// eDataMappingVarNames.Router_Mobile_ModemState: 				st_Variable:= IotExtractType(monitor.Router.Mobile.ModemState, 0, 0); 
// eDataMappingVarNames.Router_Mobile_NetworkState: 				st_Variable:= IotExtractType(monitor.Router.Mobile.NetworkState, 0, 0); 
// eDataMappingVarNames.Router_Mobile_ui_ActiveSim: 				st_Variable:= IotExtractType(monitor.Router.Mobile.ui_ActiveSim, 0, 0); 
// eDataMappingVarNames.Router_Mobile_SimStatus: 				st_Variable:= IotExtractType(monitor.Router.Mobile.SimStatus, 0, 0); 
// eDataMappingVarNames.Router_Wifi_WifiClienModeStatus: 				st_Variable:= IotExtractType(monitor.Router.Wifi.WifiClienModeStatus, 0, 0); 
// eDataMappingVarNames.Router_Wifi_WifiAPModeStatus: 				st_Variable:= IotExtractType(monitor.Router.Wifi.WifiAPModeStatus, 0, 0); 
// eDataMappingVarNames.Router_Wifi_WifiApNumberOfClients: 				st_Variable:= IotExtractType(monitor.Router.Wifi.WifiApNumberOfClients, 0, 0); 
// eDataMappingVarNames.Router_e_SMSStatus: 				st_Variable:= IotExtractType(monitor.Router.e_SMSStatus, 0, 0); 
// eDataMappingVarNames.Router_Events_b_MBCommWarning: 				st_Variable:= IotExtractType(monitor.Router.Events.b_MBCommWarning, 0, 0); 
// eDataMappingVarNames.Router_Events_b_NoSimWarning: 				st_Variable:= IotExtractType(monitor.Router.Events.b_NoSimWarning, 0, 0); 
// eDataMappingVarNames.Router_Events_b_NoNetworkWarning: 				st_Variable:= IotExtractType(monitor.Router.Events.b_NoNetworkWarning, 0, 0); 
// eDataMappingVarNames.Router_Events_b_noGPSFixWarning: 				st_Variable:= IotExtractType(monitor.Router.Events.b_noGPSFixWarning, 0, 0); 
// eDataMappingVarNames.Router_Events_b_SMSNotSendError: 				st_Variable:= IotExtractType(monitor.Router.Events.b_SMSNotSendError, 0, 0); 
// eDataMappingVarNames.Router_Events_b_NoSMSNumberAvailable: 				st_Variable:= IotExtractType(monitor.Router.Events.b_NoSMSNumberAvailable, 0, 0); 
// eDataMappingVarNames.Router_Events_b_TimeUpdateFailed: 				st_Variable:= IotExtractType(monitor.Router.Events.b_TimeUpdateFailed, 0, 0); 
// eDataMappingVarNames.controlfb_control_b_start: 															st_Variable:= IotExtractType(controlvars.control.b_start, 0, 0); 
// eDataMappingVarNames.controlfb_control_b_stop: 																st_Variable:= IotExtractType(controlvars.control.b_stop, 0, 0); 
// eDataMappingVarNames.controlfb_control_b_shutdown: 															st_Variable:= IotExtractType(controlvars.control.b_shutdown, 0, 0); 
// eDataMappingVarNames.controlfb_control_b_Reset: 															st_Variable:= IotExtractType(controlvars.control.b_Reset, 0, 0); 
// eDataMappingVarNames.controlfb_control_b_SystemShutdown: 													st_Variable:= IotExtractType(controlvars.control.b_SystemShutdown, 0, 0); 
// eDataMappingVarNames.controlfb_control_b_EMstop: 															st_Variable:= IotExtractType(controlvars.control.b_EMstop, 0, 0); 
// eDataMappingVarNames.controlfb_control_b_ClearHistory: 														st_Variable:= IotExtractType(controlvars.control.b_ClearHistory, 0, 0); 
// eDataMappingVarNames.controlfb_control_b_ActivateSettings: 													st_Variable:= IotExtractType(controlvars.control.b_ActivateSettings, 0, 0); 
// eDataMappingVarNames.controlfb_control_b_startDeHum: 														st_Variable:= IotExtractType(controlvars.control.b_startDeHum, 0, 0); 
// eDataMappingVarNames.controlfb_Operation_inputgrid_b_SyncClose: 											st_Variable:= IotExtractType(controlvars.Operation.inputgrid.b_SyncClose, 0, 0); 
// eDataMappingVarNames.controlfb_Operation_Genset_b_manualStart: 												st_Variable:= IotExtractType(controlvars.Operation.Genset.b_manualStart, 0, 0); 
// eDataMappingVarNames.controlfb_Operation_PSB_b_SyncClose: 													st_Variable:= IotExtractType(controlvars.Operation.PSB.b_SyncClose, 0, 0); 
// eDataMappingVarNames.controlfb_Operation_charger_b_StartCharging: 											st_Variable:= IotExtractType(controlvars.Operation.charger.b_StartCharging, 0, 0); 
// eDataMappingVarNames.controlfb_Operation_charger_b_ResetCharger: 											st_Variable:= IotExtractType(controlvars.Operation.charger.b_ResetCharger, 0, 0); 
// eDataMappingVarNames.controlfb_Operation_system_r_NominalVoltage: 											st_Variable:= IotExtractType(controlvars.Operation.system.r_NominalVoltage, 0, 0); 
// eDataMappingVarNames.controlfb_Operation_system_r_NominalFrequency: 										st_Variable:= IotExtractType(controlvars.Operation.system.r_NominalFrequency, 0, 0); 
// eDataMappingVarNames.controlfb_Operation_system_r_Pset: 													st_Variable:= IotExtractType(controlvars.Operation.system.r_Pset, 0, 0); 
// eDataMappingVarNames.controlfb_Operation_system_r_Qset: 													st_Variable:= IotExtractType(controlvars.Operation.system.r_Qset, 0, 0); 
// eDataMappingVarNames.controlfb_Operation_system_r_PFset: 													st_Variable:= IotExtractType(controlvars.Operation.system.r_PFset, 0, 0); 
// eDataMappingVarNames.controlfb_Operation_system_b_PFsetEnable: 												st_Variable:= IotExtractType(controlvars.Operation.system.b_PFsetEnable, 0, 0); 
// eDataMappingVarNames.controlfb_Operation_system_b_SounderMute: 												st_Variable:= IotExtractType(controlvars.Operation.system.b_SounderMute, 0, 0); 
// eDataMappingVarNames.controlfb_Operation_system_b_SounderTest: 												st_Variable:= IotExtractType(controlvars.Operation.system.b_SounderTest, 0, 0); 
// eDataMappingVarNames.controlfb_Operation_system_b_GenGridModeTrans: 										st_Variable:= IotExtractType(controlvars.Operation.system.b_GenGridModeTrans, 0, 0); 
// eDataMappingVarNames.controlfb_Operation_system_b_GridTakeOverEnable: 										st_Variable:= IotExtractType(controlvars.Operation.system.b_GridTakeOverEnable, 0, 0); 
// eDataMappingVarNames.controlfb_Operation_parallel_b_DetectSlaves: 											st_Variable:= IotExtractType(controlvars.Operation.parallel.b_DetectSlaves, 0, 0); 
// eDataMappingVarNames.controlfb_Operation_parallel_r_ActivePowerSlave1: 										st_Variable:= IotExtractType(controlvars.Operation.parallel.r_ActivePowerSlave1, 0, 0); 
// eDataMappingVarNames.controlfb_Operation_parallel_r_ReactivePowerSlave1: 									st_Variable:= IotExtractType(controlvars.Operation.parallel.r_ReactivePowerSlave1, 0, 0); 
// eDataMappingVarNames.controlfb_Operation_parallel_r_ActivePowerSlave2: 										st_Variable:= IotExtractType(controlvars.Operation.parallel.r_ActivePowerSlave2, 0, 0); 
// eDataMappingVarNames.controlfb_Operation_parallel_r_ReactivePowerSlave2: 									st_Variable:= IotExtractType(controlvars.Operation.parallel.r_ReactivePowerSlave2, 0, 0); 
// eDataMappingVarNames.controlfb_Operation_BMS_b_ManualStartHVDC: 											st_Variable:= IotExtractType(controlvars.Operation.BMS.b_ManualStartHVDC, 0, 0); 
// eDataMappingVarNames.controlfb_SoftSettings_inputgrid_PeakshaveMode: 										st_Variable:= IotExtractType(controlvars.SoftSettings.inputgrid.PeakshaveMode, 0, 0); 
// eDataMappingVarNames.controlfb_SoftSettings_inputgrid_setpointTimeslot1_r_SocTarget:		 				st_Variable:= IotExtractType(controlvars.SoftSettings.inputgrid.setpointTimeslot1.r_SocTarget, 0, 0); 
// eDataMappingVarNames.controlfb_SoftSettings_inputgrid_setpointTimeslot1_r_IdleChargePower: 					st_Variable:= IotExtractType(controlvars.SoftSettings.inputgrid.setpointTimeslot1.r_IdleChargePower, 0, 0); 
// eDataMappingVarNames.controlfb_SoftSettings_inputgrid_setpointTimeslot1_r_FeedInCurrentLimitSoft: 			st_Variable:= IotExtractType(controlvars.SoftSettings.inputgrid.setpointTimeslot1.r_FeedInCurrentLimitSoft, 0, 0); 
// eDataMappingVarNames.controlfb_SoftSettings_inputgrid_setpointTimeslot1_r_SupplyCurrentLimitSoft: 			st_Variable:= IotExtractType(controlvars.SoftSettings.inputgrid.setpointTimeslot1.r_SupplyCurrentLimitSoft, 0, 0); 
// eDataMappingVarNames.controlfb_SoftSettings_inputgrid_setpointTimeslot2_r_SocTarget: 						st_Variable:= IotExtractType(controlvars.SoftSettings.inputgrid.setpointTimeslot2.r_SocTarget, 0, 0); 
// eDataMappingVarNames.controlfb_SoftSettings_inputgrid_setpointTimeslot2_r_IdleChargePower: 					st_Variable:= IotExtractType(controlvars.SoftSettings.inputgrid.setpointTimeslot2.r_IdleChargePower, 0, 0); 
// eDataMappingVarNames.controlfb_SoftSettings_inputgrid_setpointTimeslot2_r_FeedInCurrentLimitSoft: 			st_Variable:= IotExtractType(controlvars.SoftSettings.inputgrid.setpointTimeslot2.r_FeedInCurrentLimitSoft, 0, 0); 
// eDataMappingVarNames.controlfb_SoftSettings_inputgrid_setpointTimeslot2_r_SupplyCurrentLimitSoft: 			st_Variable:= IotExtractType(controlvars.SoftSettings.inputgrid.setpointTimeslot2.r_SupplyCurrentLimitSoft, 0, 0); 
// eDataMappingVarNames.controlfb_SoftSettings_inputgrid_b_BreakerControl: 									st_Variable:= IotExtractType(controlvars.SoftSettings.inputgrid.b_BreakerControl, 0, 0); 
// eDataMappingVarNames.controlfb_SoftSettings_inputgrid_b_ReverseCTDirection: 								st_Variable:= IotExtractType(controlvars.SoftSettings.inputgrid.b_ReverseCTDirection, 0, 0); 
// eDataMappingVarNames.controlfb_SoftSettings_inputgrid_ui_CTrange: 											st_Variable:= IotExtractType(controlvars.SoftSettings.inputgrid.ui_CTrange, 0, 0); 
// eDataMappingVarNames.controlfb_SoftSettings_inputgrid_r_VTratio: 											st_Variable:= IotExtractType(controlvars.SoftSettings.inputgrid.r_VTratio, 0, 0); 
// eDataMappingVarNames.controlfb_SoftSettings_inputgrid_b_GridCodesActive: 									st_Variable:= IotExtractType(controlvars.SoftSettings.inputgrid.b_GridCodesActive, 0, 0); 
// eDataMappingVarNames.controlfb_SoftSettings_inputgrid_b_WeakGridInput: 										st_Variable:= IotExtractType(controlvars.SoftSettings.inputgrid.b_WeakGridInput, 0, 0); 
// eDataMappingVarNames.controlfb_SoftSettings_inputgrid_breaker_AutoConnect: 									st_Variable:= IotExtractType(controlvars.SoftSettings.inputgrid.breaker.AutoConnect, 0, 0); 
// eDataMappingVarNames.controlfb_SoftSettings_inputgrid_breaker_ShutdownDisconnect: 							st_Variable:= IotExtractType(controlvars.SoftSettings.inputgrid.breaker.ShutdownDisconnect, 0, 0); 
// eDataMappingVarNames.controlfb_SoftSettings_inputgrid_breaker_EMstopDisconnect: 							st_Variable:= IotExtractType(controlvars.SoftSettings.inputgrid.breaker.EMstopDisconnect, 0, 0); 
// eDataMappingVarNames.controlfb_SoftSettings_inputgrid_breaker_CurrentLimitDisconnect: 						st_Variable:= IotExtractType(controlvars.SoftSettings.inputgrid.breaker.CurrentLimitDisconnect, 0, 0); 
// eDataMappingVarNames.controlfb_SoftSettings_inputgrid_breaker_CurrentLimitRetries: 							st_Variable:= IotExtractType(controlvars.SoftSettings.inputgrid.breaker.CurrentLimitRetries, 0, 0); 
// eDataMappingVarNames.controlfb_SoftSettings_inputgenset_b_AutoStartStop: 									st_Variable:= IotExtractType(controlvars.SoftSettings.inputgenset.b_AutoStartStop, 0, 0); 
// eDataMappingVarNames.controlfb_SoftSettings_inputgenset_b_HydridMode: 										st_Variable:= IotExtractType(controlvars.SoftSettings.inputgenset.b_HydridMode, 0, 0); 
// eDataMappingVarNames.controlfb_SoftSettings_inputgenset_b_EnableSchedule: 									st_Variable:= IotExtractType(controlvars.SoftSettings.inputgenset.b_EnableSchedule, 0, 0); 
// eDataMappingVarNames.controlfb_SoftSettings_inputgenset_setpointTimeslot1_r_SoCStart: 						st_Variable:= IotExtractType(controlvars.SoftSettings.inputgenset.setpointTimeslot1.r_SoCStart, 0, 0); 
// eDataMappingVarNames.controlfb_SoftSettings_inputgenset_setpointTimeslot1_r_SoCStop: 						st_Variable:= IotExtractType(controlvars.SoftSettings.inputgenset.setpointTimeslot1.r_SoCStop, 0, 0); 
// eDataMappingVarNames.controlfb_SoftSettings_inputgenset_setpointTimeslot1_r_BatteryloadStart: 				st_Variable:= IotExtractType(controlvars.SoftSettings.inputgenset.setpointTimeslot1.r_BatteryloadStart, 0, 0); 
// eDataMappingVarNames.controlfb_SoftSettings_inputgenset_setpointTimeslot1_r_BatteryloadStop: 				st_Variable:= IotExtractType(controlvars.SoftSettings.inputgenset.setpointTimeslot1.r_BatteryloadStop, 0, 0); 
// eDataMappingVarNames.controlfb_SoftSettings_inputgenset_setpointTimeslot1_b_StartAtBatteryError: 			st_Variable:= IotExtractType(controlvars.SoftSettings.inputgenset.setpointTimeslot1.b_StartAtBatteryError, 0, 0); 
// eDataMappingVarNames.controlfb_SoftSettings_inputgenset_setpointTimeslot2_r_SoCStart: 						st_Variable:= IotExtractType(controlvars.SoftSettings.inputgenset.setpointTimeslot2.r_SoCStart, 0, 0); 
// eDataMappingVarNames.controlfb_SoftSettings_inputgenset_setpointTimeslot2_r_SoCStop: 						st_Variable:= IotExtractType(controlvars.SoftSettings.inputgenset.setpointTimeslot2.r_SoCStop, 0, 0); 
// eDataMappingVarNames.controlfb_SoftSettings_inputgenset_setpointTimeslot2_r_BatteryloadStart: 				st_Variable:= IotExtractType(controlvars.SoftSettings.inputgenset.setpointTimeslot2.r_BatteryloadStart, 0, 0); 
// eDataMappingVarNames.controlfb_SoftSettings_inputgenset_setpointTimeslot2_r_BatteryloadStop: 				st_Variable:= IotExtractType(controlvars.SoftSettings.inputgenset.setpointTimeslot2.r_BatteryloadStop, 0, 0); 
// eDataMappingVarNames.controlfb_SoftSettings_inputgenset_setpointTimeslot2_b_StartAtBatteryError: 			st_Variable:= IotExtractType(controlvars.SoftSettings.inputgenset.setpointTimeslot2.b_StartAtBatteryError, 0, 0); 
// eDataMappingVarNames.controlfb_SoftSettings_inputgenset_b_PSBExtGensetMonitoring: 							st_Variable:= IotExtractType(controlvars.SoftSettings.inputgenset.b_PSBExtGensetMonitoring, 0, 0); 
// eDataMappingVarNames.controlfb_SoftSettings_inputgenset_b_FreqProtectionEnable: 							st_Variable:= IotExtractType(controlvars.SoftSettings.inputgenset.b_FreqProtectionEnable, 0, 0); 
// eDataMappingVarNames.controlfb_SoftSettings_inputgenset_Generator_e_GensetMode: 							st_Variable:= IotExtractType(controlvars.SoftSettings.inputgenset.Generator.e_GensetMode, 0, 0); 
// eDataMappingVarNames.controlfb_SoftSettings_inputgenset_Generator_b_GensetLoadshareLine: 					st_Variable:= IotExtractType(controlvars.SoftSettings.inputgenset.Generator.b_GensetLoadshareLine, 0, 0); 
// eDataMappingVarNames.controlfb_SoftSettings_inputgenset_Generator_r_RatedPower: 							st_Variable:= IotExtractType(controlvars.SoftSettings.inputgenset.Generator.r_RatedPower, 0, 0); 
// eDataMappingVarNames.controlfb_SoftSettings_inputgenset_Generator_r_powerloadMax: 							st_Variable:= IotExtractType(controlvars.SoftSettings.inputgenset.Generator.r_powerloadMax, 0, 0); 
// eDataMappingVarNames.controlfb_SoftSettings_inputgenset_Generator_r_PowerloadMin: 							st_Variable:= IotExtractType(controlvars.SoftSettings.inputgenset.Generator.r_PowerloadMin, 0, 0); 
// eDataMappingVarNames.controlfb_SoftSettings_inputgenset_Generator_r_PowerloadEff: 							st_Variable:= IotExtractType(controlvars.SoftSettings.inputgenset.Generator.r_PowerloadEff, 0, 0); 
// eDataMappingVarNames.controlfb_SoftSettings_inputgenset_Generator_r_ramprate: 								st_Variable:= IotExtractType(controlvars.SoftSettings.inputgenset.Generator.r_ramprate, 0, 0); 
// eDataMappingVarNames.controlfb_SoftSettings_inputgenset_Generator_ui_CooldownTime: 							st_Variable:= IotExtractType(controlvars.SoftSettings.inputgenset.Generator.ui_CooldownTime, 0, 0); 
// eDataMappingVarNames.controlfb_SoftSettings_inputgenset_Generator_ui_WarmupTime: 							st_Variable:= IotExtractType(controlvars.SoftSettings.inputgenset.Generator.ui_WarmupTime, 0, 0); 
// eDataMappingVarNames.controlfb_SoftSettings_inputgenset_Loadbank_b_Enable: 									st_Variable:= IotExtractType(controlvars.SoftSettings.inputgenset.Loadbank.b_Enable, 0, 0); 
// eDataMappingVarNames.controlfb_SoftSettings_inputgenset_Loadbank_r_PowerRating: 							st_Variable:= IotExtractType(controlvars.SoftSettings.inputgenset.Loadbank.r_PowerRating, 0, 0); 
// eDataMappingVarNames.controlfb_SoftSettings_inputgenset_Loadbank_r_PowerStepSize: 							st_Variable:= IotExtractType(controlvars.SoftSettings.inputgenset.Loadbank.r_PowerStepSize, 0, 0); 
// eDataMappingVarNames.controlfb_SoftSettings_PSB_PeakshaveMode: 												st_Variable:= IotExtractType(controlvars.SoftSettings.PSB.PeakshaveMode, 0, 0); 
// eDataMappingVarNames.controlfb_SoftSettings_PSB_setpointTimeslot1_r_SocTarget: 								st_Variable:= IotExtractType(controlvars.SoftSettings.PSB.setpointTimeslot1.r_SocTarget, 0, 0); 
// eDataMappingVarNames.controlfb_SoftSettings_PSB_setpointTimeslot1_r_IdleChargePower: 						st_Variable:= IotExtractType(controlvars.SoftSettings.PSB.setpointTimeslot1.r_IdleChargePower, 0, 0); 
// eDataMappingVarNames.controlfb_SoftSettings_PSB_setpointTimeslot1_r_FeedInCurrentLimitSoft: 				st_Variable:= IotExtractType(controlvars.SoftSettings.PSB.setpointTimeslot1.r_FeedInCurrentLimitSoft, 0, 0); 
// eDataMappingVarNames.controlfb_SoftSettings_PSB_setpointTimeslot1_r_SupplyCurrentLimitSoft: 				st_Variable:= IotExtractType(controlvars.SoftSettings.PSB.setpointTimeslot1.r_SupplyCurrentLimitSoft, 0, 0); 
// eDataMappingVarNames.controlfb_SoftSettings_PSB_setpointTimeslot2_r_SocTarget: 								st_Variable:= IotExtractType(controlvars.SoftSettings.PSB.setpointTimeslot2.r_SocTarget, 0, 0); 
// eDataMappingVarNames.controlfb_SoftSettings_PSB_setpointTimeslot2_r_IdleChargePower: 						st_Variable:= IotExtractType(controlvars.SoftSettings.PSB.setpointTimeslot2.r_IdleChargePower, 0, 0); 
// eDataMappingVarNames.controlfb_SoftSettings_PSB_setpointTimeslot2_r_FeedInCurrentLimitSoft: 				st_Variable:= IotExtractType(controlvars.SoftSettings.PSB.setpointTimeslot2.r_FeedInCurrentLimitSoft, 0, 0); 
// eDataMappingVarNames.controlfb_SoftSettings_PSB_setpointTimeslot2_r_SupplyCurrentLimitSoft: 				st_Variable:= IotExtractType(controlvars.SoftSettings.PSB.setpointTimeslot2.r_SupplyCurrentLimitSoft, 0, 0); 
// eDataMappingVarNames.controlfb_SoftSettings_PSB_b_BreakerControl: 											st_Variable:= IotExtractType(controlvars.SoftSettings.PSB.b_BreakerControl, 0, 0); 
// eDataMappingVarNames.controlfb_SoftSettings_PSB_b_ReverseCTDirection: 										st_Variable:= IotExtractType(controlvars.SoftSettings.PSB.b_ReverseCTDirection, 0, 0); 
// eDataMappingVarNames.controlfb_SoftSettings_PSB_ui_CTrange: 												st_Variable:= IotExtractType(controlvars.SoftSettings.PSB.ui_CTrange, 0, 0); 
// eDataMappingVarNames.controlfb_SoftSettings_PSB_r_VTratio: 													st_Variable:= IotExtractType(controlvars.SoftSettings.PSB.r_VTratio, 0, 0); 
// eDataMappingVarNames.controlfb_SoftSettings_system_b_EnableSchedule: 										st_Variable:= IotExtractType(controlvars.SoftSettings.system.b_EnableSchedule, 0, 0); 
// eDataMappingVarNames.controlfb_SoftSettings_system_b_EnableTransportMode: 									st_Variable:= IotExtractType(controlvars.SoftSettings.system.b_EnableTransportMode, 0, 0); 
// eDataMappingVarNames.controlfb_SoftSettings_system_b_EcoModeEnable: 										st_Variable:= IotExtractType(controlvars.SoftSettings.system.b_EcoModeEnable, 0, 0); 
// eDataMappingVarNames.controlfb_SoftSettings_system_e_UgridPowerMode: 										st_Variable:= IotExtractType(controlvars.SoftSettings.system.e_UgridPowerMode, 0, 0); 
// eDataMappingVarNames.controlfb_SoftSettings_system_e_NetcontactorMode: 										st_Variable:= IotExtractType(controlvars.SoftSettings.system.e_NetcontactorMode, 0, 0); 
// eDataMappingVarNames.controlfb_SoftSettings_system_e_UgridPowerLimitingMode: 								st_Variable:= IotExtractType(controlvars.SoftSettings.system.e_UgridPowerLimitingMode, 0, 0); 
// eDataMappingVarNames.controlfb_SoftSettings_system_b_AutomaticSwitching: 									st_Variable:= IotExtractType(controlvars.SoftSettings.system.b_AutomaticSwitching, 0, 0); 
// eDataMappingVarNames.controlfb_SoftSettings_system_b_AMF: 													st_Variable:= IotExtractType(controlvars.SoftSettings.system.b_AMF, 0, 0); 
// eDataMappingVarNames.controlfb_SoftSettings_system_r_FrequencyDroop: 										st_Variable:= IotExtractType(controlvars.SoftSettings.system.r_FrequencyDroop, 0, 0); 
// eDataMappingVarNames.controlfb_SoftSettings_system_r_VoltageDroop: 											st_Variable:= IotExtractType(controlvars.SoftSettings.system.r_VoltageDroop, 0, 0); 
// eDataMappingVarNames.controlfb_SoftSettings_system_r_SocMin: 												st_Variable:= IotExtractType(controlvars.SoftSettings.system.r_SocMin, 0, 0); 
// eDataMappingVarNames.controlfb_SoftSettings_system_r_SocMax: 												st_Variable:= IotExtractType(controlvars.SoftSettings.system.r_SocMax, 0, 0); 
// eDataMappingVarNames.controlfb_SoftSettings_system_r_PDischargeLimit: 										st_Variable:= IotExtractType(controlvars.SoftSettings.system.r_PDischargeLimit, 0, 0); 
// eDataMappingVarNames.controlfb_SoftSettings_system_r_PChargeLimit: 											st_Variable:= IotExtractType(controlvars.SoftSettings.system.r_PChargeLimit, 0, 0); 
// eDataMappingVarNames.controlfb_SoftSettings_system_r_AMax: 													st_Variable:= IotExtractType(controlvars.SoftSettings.system.r_AMax, 0, 0); 
// eDataMappingVarNames.controlfb_SoftSettings_system_s_SystemName: 											st_Variable:= IotExtractType(controlvars.SoftSettings.system.s_SystemName, 0, 0); 
// eDataMappingVarNames.controlfb_SoftSettings_system_s_SMSnumber: 											st_Variable:= IotExtractType(controlvars.SoftSettings.system.s_SMSnumber, 0, 0); 
// eDataMappingVarNames.controlfb_SoftSettings_system_ScheduleTimeSlot1_b_active: 								st_Variable:= IotExtractType(controlvars.SoftSettings.system.ScheduleTimeSlot1.b_active, 0, 0); 
// eDataMappingVarNames.controlfb_SoftSettings_system_ScheduleTimeSlot1_usi_DayOfWeek: 						st_Variable:= IotExtractType(controlvars.SoftSettings.system.ScheduleTimeSlot1.usi_DayOfWeek, 0, 0); 
// eDataMappingVarNames.controlfb_SoftSettings_system_ScheduleTimeSlot1_usi_HourOfDay: 						st_Variable:= IotExtractType(controlvars.SoftSettings.system.ScheduleTimeSlot1.usi_HourOfDay, 0, 0); 
// eDataMappingVarNames.controlfb_SoftSettings_system_ScheduleTimeSlot1_usi_MinuteOfHour: 						st_Variable:= IotExtractType(controlvars.SoftSettings.system.ScheduleTimeSlot1.usi_MinuteOfHour, 0, 0); 
// eDataMappingVarNames.controlfb_SoftSettings_system_ScheduleTimeSlot2_b_active: 								st_Variable:= IotExtractType(controlvars.SoftSettings.system.ScheduleTimeSlot2.b_active, 0, 0); 
// eDataMappingVarNames.controlfb_SoftSettings_system_ScheduleTimeSlot2_usi_DayOfWeek: 						st_Variable:= IotExtractType(controlvars.SoftSettings.system.ScheduleTimeSlot2.usi_DayOfWeek, 0, 0); 
// eDataMappingVarNames.controlfb_SoftSettings_system_ScheduleTimeSlot2_usi_HourOfDay: 						st_Variable:= IotExtractType(controlvars.SoftSettings.system.ScheduleTimeSlot2.usi_HourOfDay, 0, 0); 
// eDataMappingVarNames.controlfb_SoftSettings_system_ScheduleTimeSlot2_usi_MinuteOfHour: 						st_Variable:= IotExtractType(controlvars.SoftSettings.system.ScheduleTimeSlot2.usi_MinuteOfHour, 0, 0); 
// eDataMappingVarNames.controlfb_SoftSettings_system_by_LEDbrightness: 										st_Variable:= IotExtractType(controlvars.SoftSettings.system.by_LEDbrightness, 0, 0); 
// eDataMappingVarNames.controlfb_SoftSettings_setup_e_AcInputType: 											st_Variable:= IotExtractType(controlvars.SoftSettings.setup.e_AcInputType, 0, 0); 
// eDataMappingVarNames.controlfb_SoftSettings_setup_b_MasterSlaveMode: 										st_Variable:= IotExtractType(controlvars.SoftSettings.setup.b_MasterSlaveMode, 0, 0); 
// eDataMappingVarNames.controlfb_SoftSettings_setup_b_PeakshaveBoxEnable: 									st_Variable:= IotExtractType(controlvars.SoftSettings.setup.b_PeakshaveBoxEnable, 0, 0); 
// eDataMappingVarNames.controlfb_SoftSettings_setup_e_Gridmode: 												st_Variable:= IotExtractType(controlvars.SoftSettings.setup.e_Gridmode, 0, 0); 
// eDataMappingVarNames.controlfb_SoftSettings_setup_e_DcCouplingType: 										st_Variable:= IotExtractType(controlvars.SoftSettings.setup.e_DcCouplingType, 0, 0); 
// eDataMappingVarNames.controlfb_SoftSettings_setup_b_ExtGenset: 												st_Variable:= IotExtractType(controlvars.SoftSettings.setup.b_ExtGenset, 0, 0); 
// eDataMappingVarNames.controlfb_HardSettings_setup_e_ControlSource: 											st_Variable:= IotExtractType(controlvars.HardSettings.setup.e_ControlSource, 0, 0); 
// eDataMappingVarNames.controlfb_HardSettings_charger_r_PowerMax: 											st_Variable:= IotExtractType(controlvars.HardSettings.charger.r_PowerMax, 0, 0); 
// eDataMappingVarNames.controlfb_HardSettings_parallel_b_MasterSlaveEnabled: 									st_Variable:= IotExtractType(controlvars.HardSettings.parallel.b_MasterSlaveEnabled, 0, 0); 
// eDataMappingVarNames.controlfb_HardSettings_parallel_b_UnitIsMaster: 										st_Variable:= IotExtractType(controlvars.HardSettings.parallel.b_UnitIsMaster, 0, 0); 
// eDataMappingVarNames.controlfb_HardSettings_parallel_b_ShutdownOnCommError: 								st_Variable:= IotExtractType(controlvars.HardSettings.parallel.b_ShutdownOnCommError, 0, 0); 
// eDataMappingVarNames.controlfb_HardSettings_parallel_b_EffiencyMode: 										st_Variable:= IotExtractType(controlvars.HardSettings.parallel.b_EffiencyMode, 0, 0); 
// eDataMappingVarNames.controlfb_HardSettings_parallel_r_VoltageDroop: 										st_Variable:= IotExtractType(controlvars.HardSettings.parallel.r_VoltageDroop, 0, 0); 
// eDataMappingVarNames.controlfb_HardSettings_parallel_r_FrequencyDroop: 										st_Variable:= IotExtractType(controlvars.HardSettings.parallel.r_FrequencyDroop, 0, 0); 
// eDataMappingVarNames.controlfb_HardSettings_system_r_PDischargeLimit: 										st_Variable:= IotExtractType(controlvars.HardSettings.system.r_PDischargeLimit, 0, 0); 
// eDataMappingVarNames.controlfb_HardSettings_system_r_PChargeLimit: 											st_Variable:= IotExtractType(controlvars.HardSettings.system.r_PChargeLimit, 0, 0); 
// eDataMappingVarNames.controlfb_HardSettings_system_r_SMax: 													st_Variable:= IotExtractType(controlvars.HardSettings.system.r_SMax, 0, 0); 
// eDataMappingVarNames.controlfb_HardSettings_system_r_Amax: 													st_Variable:= IotExtractType(controlvars.HardSettings.system.r_Amax, 0, 0); 
// eDataMappingVarNames.controlfb_HardSettings_system_e_EarthingSystem: 										st_Variable:= IotExtractType(controlvars.HardSettings.system.e_EarthingSystem, 0, 0); 
// eDataMappingVarNames.controlfb_HardSettings_system_a_ui_InputCurrentLimit_1: 								st_Variable:= IotExtractType(controlvars.HardSettings.system.a_ui_InputCurrentLimit[1], 0, 0); 
// eDataMappingVarNames.controlfb_HardSettings_system_a_ui_InputCurrentLimit_2: 								st_Variable:= IotExtractType(controlvars.HardSettings.system.a_ui_InputCurrentLimit[2], 0, 0); 
// eDataMappingVarNames.controlfb_HardSettings_system_a_ui_OutputCurrentLimit_1: 								st_Variable:= IotExtractType(controlvars.HardSettings.system.a_ui_OutputCurrentLimit[1], 0, 0); 
// eDataMappingVarNames.controlfb_HardSettings_system_a_ui_OutputCurrentLimit_2: 								st_Variable:= IotExtractType(controlvars.HardSettings.system.a_ui_OutputCurrentLimit[2], 0, 0); 
// eDataMappingVarNames.controlfb_HardSettings_system_a_ui_OutputCurrentLimit_3: 								st_Variable:= IotExtractType(controlvars.HardSettings.system.a_ui_OutputCurrentLimit[3], 0, 0); 
// eDataMappingVarNames.Generator_CommunicationOK: 				st_Variable:= IotExtractType(monitor.Generator.CommunicationOK, 0, 0); 
// eDataMappingVarNames.Generator_FuelLow: 				st_Variable:= IotExtractType(monitor.Generator.FuelLow, 0, 0); 
// eDataMappingVarNames.Generator_FuelCritical: 				st_Variable:= IotExtractType(monitor.Generator.FuelCritical, 0, 0); 
// eDataMappingVarNames.Generator_bGenBreakerClosed: 				st_Variable:= IotExtractType(monitor.Generator.bGenBreakerClosed, 0, 0); 
// eDataMappingVarNames.Generator_bMainBreakerClosed: 				st_Variable:= IotExtractType(monitor.Generator.bMainBreakerClosed, 0, 0); 
// eDataMappingVarNames.Generator_bGenRunning: 				st_Variable:= IotExtractType(monitor.Generator.bGenRunning, 0, 0); 
// eDataMappingVarNames.Generator_bGenVoltFreqOK: 				st_Variable:= IotExtractType(monitor.Generator.bGenVoltFreqOK, 0, 0); 
// eDataMappingVarNames.Generator_bMainsFailure: 				st_Variable:= IotExtractType(monitor.Generator.bMainsFailure, 0, 0); 
// eDataMappingVarNames.Generator_eActiveGenMode: 				st_Variable:= IotExtractType(monitor.Generator.eActiveGenMode, 0, 0); 
// eDataMappingVarNames.Generator_bIslandModeActive: 				st_Variable:= IotExtractType(monitor.Generator.bIslandModeActive, 0, 0); 
// eDataMappingVarNames.Generator_bAMFActive: 				st_Variable:= IotExtractType(monitor.Generator.bAMFActive, 0, 0); 
// eDataMappingVarNames.Generator_bPeakshaveActive: 				st_Variable:= IotExtractType(monitor.Generator.bPeakshaveActive, 0, 0); 
// eDataMappingVarNames.Generator_bFixedPowerActive: 				st_Variable:= IotExtractType(monitor.Generator.bFixedPowerActive, 0, 0); 
// eDataMappingVarNames.Generator_ar_LineVoltage_AVG: 				st_Variable:= IotExtractType(monitor.Generator.ar_LineVoltage[0], 1, 1); 
// eDataMappingVarNames.Generator_ar_LineVoltage_L1: 				st_Variable:= IotExtractType(monitor.Generator.ar_LineVoltage[1], 1, 1); 
// eDataMappingVarNames.Generator_ar_LineVoltage_L2: 				st_Variable:= IotExtractType(monitor.Generator.ar_LineVoltage[2], 1, 1); 
// eDataMappingVarNames.Generator_ar_LineVoltage_L3: 				st_Variable:= IotExtractType(monitor.Generator.ar_LineVoltage[3], 1, 1); 
// eDataMappingVarNames.Generator_ar_PhaseVoltage_AVG: 				st_Variable:= IotExtractType(monitor.Generator.ar_PhaseVoltage[0], 1, 1); 
// eDataMappingVarNames.Generator_ar_PhaseVoltage_L1: 				st_Variable:= IotExtractType(monitor.Generator.ar_PhaseVoltage[1], 1, 1); 
// eDataMappingVarNames.Generator_ar_PhaseVoltage_L2: 				st_Variable:= IotExtractType(monitor.Generator.ar_PhaseVoltage[2], 1, 1); 
// eDataMappingVarNames.Generator_ar_PhaseVoltage_L3: 				st_Variable:= IotExtractType(monitor.Generator.ar_PhaseVoltage[3], 1, 1); 
// eDataMappingVarNames.Generator_ar_Frequency_AVG: 				st_Variable:= IotExtractType(monitor.Generator.ar_Frequency[0], 2, 1); 
// eDataMappingVarNames.Generator_ar_Frequency_L1: 				st_Variable:= IotExtractType(monitor.Generator.ar_Frequency[1], 2, 1); 
// eDataMappingVarNames.Generator_ar_Frequency_L2: 				st_Variable:= IotExtractType(monitor.Generator.ar_Frequency[2], 2, 1); 
// eDataMappingVarNames.Generator_ar_Frequency_L3: 				st_Variable:= IotExtractType(monitor.Generator.ar_Frequency[3], 2, 1); 
// eDataMappingVarNames.Generator_ar_Current_AVG: 				st_Variable:= IotExtractType(monitor.Generator.ar_Current[0], 1, 1); 
// eDataMappingVarNames.Generator_ar_Current_L1: 				st_Variable:= IotExtractType(monitor.Generator.ar_Current[1], 1, 1); 
// eDataMappingVarNames.Generator_ar_Current_L2: 				st_Variable:= IotExtractType(monitor.Generator.ar_Current[2], 1, 1); 
// eDataMappingVarNames.Generator_ar_Current_L3: 				st_Variable:= IotExtractType(monitor.Generator.ar_Current[3], 1, 1); 
// eDataMappingVarNames.Generator_ar_PowerFactor_AVG: 				st_Variable:= IotExtractType(monitor.Generator.ar_PowerFactor[0], 2, 0); 
// eDataMappingVarNames.Generator_ar_ActivePower_AVG: 				st_Variable:= IotExtractType(monitor.Generator.ar_ActivePower[0], 1, 1); 
// eDataMappingVarNames.Generator_ar_ActivePower_L1: 				st_Variable:= IotExtractType(monitor.Generator.ar_ActivePower[1], 1, 1); 
// eDataMappingVarNames.Generator_ar_ActivePower_L2: 				st_Variable:= IotExtractType(monitor.Generator.ar_ActivePower[2], 1, 1); 
// eDataMappingVarNames.Generator_ar_ActivePower_L3: 				st_Variable:= IotExtractType(monitor.Generator.ar_ActivePower[3], 1, 1); 
// eDataMappingVarNames.Generator_ar_ReactivePower_AVG: 				st_Variable:= IotExtractType(monitor.Generator.ar_ReactivePower[0], 1, 1); 
// eDataMappingVarNames.Generator_ar_ApparentPower_AVG: 				st_Variable:= IotExtractType(monitor.Generator.ar_ApparentPower[0], 1, 1); 
// eDataMappingVarNames.HartingIO_b_DigitalInput1Active: 				st_Variable:= IotExtractType(monitor.HartingIO.b_DigitalInput1Active, 0, 0); 
// eDataMappingVarNames.HartingIO_b_DigitalInput2Active: 				st_Variable:= IotExtractType(monitor.HartingIO.b_DigitalInput2Active, 0, 0); 
// eDataMappingVarNames.HartingIO_b_GenLowFuel: 				st_Variable:= IotExtractType(monitor.HartingIO.b_GenLowFuel, 0, 0); 
// eDataMappingVarNames.HartingIO_b_ExtSystemShutdownRequest: 				st_Variable:= IotExtractType(monitor.HartingIO.b_ExtSystemShutdownRequest, 0, 0); 
// eDataMappingVarNames.HartingIO_b_ExtEMstopOK: 				st_Variable:= IotExtractType(monitor.HartingIO.b_ExtEMstopOK, 0, 0); 
// eDataMappingVarNames.HartingIO_b_ExtEMstopActive: 				st_Variable:= IotExtractType(monitor.HartingIO.b_ExtEMstopActive, 0, 0); 
END_CASE

IF index >= eDataMappingVarNames.controlfb_control_b_start AND index <= eDataMappingVarNames.controlfb_HardSettings_system_a_ui_OutputCurrentLimit_3 THEN
	st_RW.ReadFromNUC := aData[index].LogType <> 0;
	st_RW.WriteToNUC := FALSE;
ELSE
	st_RW.ReadFromNUC := FALSE;
	st_RW.WriteToNUC :=  aData[index].LogType <> 0;
END_IF


//-------------------------------Write to output---------------------------------------------
IotMappingV2.sName		:= aData[index].Label;				//Name of the variable
IotMappingV2.sValue		:= st_Variable.sValue;	//Extracted value of the variable
IotMappingV2.eUpdate	:= aData[index].LogInterval;				//Update frequency
IotMappingV2.st_RW		:= st_RW;				//Read/Write
IotMappingV2.pAdress	:= st_Variable.pAdress; //Adress pointer to variable
IotMappingV2.diSize		:= st_Variable.diSize;
IotMappingV2.ClassType	:= st_Variable.ClassType; //Extracted data type of the variable
IotMappingV2.bNumber	:= st_Variable.bNumber;
IotMappingV2.bJson		:= bJson;
END_METHOD

METHOD IoTWriteBacktoVar : BOOL;
VAR_INPUT
	sValue	  : STRING; //Content of variable to write to in STRING type
	pAdress	  : PVOID; //Adress of the Variable
	ClassType : __SYSTEM.TYPE_CLASS; //Type of the Variable
END_VAR

VAR
	pBool	: POINTER TO BOOL;
	pInt	: POINTER TO INT;
	pLreal	: POINTER TO LREAL;
	pWord	: POINTER TO WORD;
	pDword	: POINTER TO DWORD;
	pSint	: POINTER TO SINT;
	pReal	: POINTER TO REAL;
	pString : POINTER TO STRING;
END_VAR
CASE ClassType OF
    __SYSTEM.Type_Class.TYPE_BOOL :
		pBool:=pAdress;
		pBool^:=STRING_TO_BOOL(sValue);
    __SYSTEM.Type_Class.TYPE_ENUM :
		pInt:=pAdress;
		pInt^:=STRING_TO_INT(sValue);
    __SYSTEM.Type_Class.TYPE_LREAL :
		pLreal:=pAdress;
		pLreal^:=STRING_TO_LREAL(sValue);
    __SYSTEM.Type_Class.TYPE_WORD :
		pWord:=pAdress;
		pWord^:= STRING_TO_WORD(sValue);
    __SYSTEM.Type_Class.TYPE_DWORD :
		pDword:=pAdress;
		pDWord^:= STRING_TO_WORD(sValue);
    __SYSTEM.Type_Class.TYPE_SINT :
		pSint:=pAdress;
		pSint^:= STRING_TO_SINT(sValue);
    __SYSTEM.Type_Class.TYPE_INT :
		pInt:=pAdress;
		pInt^:=STRING_TO_INT(sValue);
    __SYSTEM.Type_Class.TYPE_REAL :
		pReal:=pAdress;
		pReal^:=STRING_TO_REAL(sValue);
    __SYSTEM.Type_Class.TYPE_STRING :	
		pString:=pAdress;
		pString^:=sValue;
		
	ELSE
		IoTWriteBackToVar:=FALSE;
END_CASE
END_METHOD

METHOD OrPublish : BOOL

VAR_INPUT
	iotprops 		: REFERENCE TO ST_IotProps;
	sOrPubPrefix	: STRING;
	sAssetID		: STRING;
END_VAR

VAR
	sTopic			: 	STRING;
	sQuote			:	STRING := '"';
END_VAR
//Prepare Topic		
sTopic:= concat(sORPubPrefix,IotProps.sName);
sTopic:= concat(sTopic,sAssetID);

//Catch NANs
IF IotProps.sValue = '#NaN' THEN
	IotProps.sValue:='0';
END_IF

//Convert payload to JSON string if text ( "sValue" )
IF NOT IotProps.bNumber AND NOT IotProps.bJson THEN
	concat2(ADR(sQuote), ADR(IotProps.sValue), ADR(IotProps.sValue), SIZEOF(IotProps.sValue));
	concat2(ADR(IotProps.sValue), ADR(sQuote), ADR(IotProps.sValue), SIZEOF(IotProps.sValue));
END_IF

//Publish 
fbMqttClient.Publish(sTopic:=sTopic,
pPayload := ADR(IotProps.sValue), //ADR(MessageToPublishJson),
nPayloadSize := LEN2(ADR(IotProps.sValue)), // ADR(MessageToPublishJson)),
eQoS := TcIotMqttQos.AtMostOnceDelivery,
bRetain:= FALSE,
bQueue := FALSE);
END_METHOD

METHOD PublishVarsV1 : BOOL
VAR_INPUT
END_VAR
b_UpdateActive := fbSendFastMessageTimer.Q OR fbSendSlowMessageTimer.Q OR bInitiateFirstTimeSend;
IF e_state = eConnectionState.authorized AND b_UpdateActive THEN
	FOR i:= 1 TO iSizeIotMappingV1 BY 1 DO	
			
		//----Get variable mapping properties corresponding to index
		st_IotProps:= IotMapping(i);
		
		//----Fast Message Sending
		IF (st_IotProps.eUpdate = eUpdate.Fast) AND st_IotProps.st_RW.WriteToNUC AND fbSendFastMessageTimer.Q THEN
				//Publish in OpenRemote format
				OrPublish(sOrPubPrefix:=sPubPrefix, sAssetID:=sAssetID, iotprops := st_IotProps);	
				//OrPublish(sOrPubPrefix:=sPubPrefix,sName:=st_IotProps.sName,sAssetID:=sAssetID,sValue:=st_IotProps.sValue, bNumber:=st_IotProps.bNumber);	
		END_IF
		
		//----Slow Message Sending---------
		IF (st_IotProps.eUpdate = eUpdate.Slow) AND st_IotProps.st_RW.WriteToNUC AND fbSendSlowMessageTimer.Q THEN		
				//Publish in OpenRemote format
				OrPublish(sOrPubPrefix:=sPubPrefix, sAssetID:=sAssetID, iotprops := st_IotProps);
		END_IF
		
		//----Maintenance Message Sending (sends every reconnect, which is reset daily)---------
		IF (st_IotProps.eUpdate = eUpdate.Daily) AND st_IotProps.st_RW.WriteToNUC AND bInitiateFirstTimeSend THEN		
				//Publish in OpenRemote format
				OrPublish(sOrPubPrefix:=sPubPrefix, sAssetID:=sAssetID, iotprops := st_IotProps);
		END_IF
		
		//----On change Message Sending------
		IF (st_IotProps.eUpdate = eUpdate.OnChange) AND st_IotProps.st_RW.WriteToNUC AND (fbSendFastMessageTimer.Q  OR bInitiateFirstTimeSend) THEN
			i_OnChangeValuesIndex := i_OnChangeValuesIndex + 1;
			
			//Evaluate whether value has changed or first time message trigger is active
			IF st_IotProps.sValue <> aPreviousValue[i_OnChangeValuesIndex] OR bInitiateFirstTimeSend THEN
				//Set current value to memory
				aPreviousValue[i_OnChangeValuesIndex]:= st_IotProps.sValue;
				//Publish in OpenRemote format
				OrPublish(sOrPubPrefix:=sPubPrefix, sAssetID:=sAssetID, iotprops := st_IotProps);

			END_IF
		END_IF	
	END_FOR
	i_OnChangeValuesIndex := 0;
	//Disable First Time send
	bInitiateFirstTimeSend:=FALSE;
END_IF
END_METHOD

METHOD PublishVarsV2 : BOOL
VAR_INPUT
	Authorized : BOOL;
	Interval : eUpdate;
END_VAR

VAR_IN_OUT
	state : ST_IOT_SentStateLog;
END_VAR

VAR
	Checksum : WORD;
	i : INT;
	Update : BOOL;
	CheckSumWordLast	: WORD;
END_VAR
IF Authorized AND State.bUpdate THEN
	State.bMessageSent := FALSE;
	FOR i:= State.LastIndexSent TO State.LastIndex BY 1 DO	
		//----Get variable mapping properties corresponding to index
//FIX MappingV2		//st_IotProps:= IotMappingV2(i);

		//---- Message Sending
		IF (st_IotProps.eUpdate = interval) AND st_IotProps.st_RW.WriteToNUC AND State.bUpdate THEN
			//Publish in OpenRemote format
			IF State.LastIndexSent < i THEN
				// onchange detection
				IF st_IotProps.eUpdate = eUpdate.OnChange THEN 
					CheckSum 	:= F_CheckSum16(st_IotProps.pAdress, st_iotProps.diSize, 0);
					Update := aCheckSumLast[i] <> CheckSum;
					aCheckSumLast[i] := CheckSum;
				ELSE
					Update := TRUE;
				END_IF
				
				//Update variable
				IF update THEN
					OrPublish(sOrPubPrefix:=sPubPrefix, sAssetID:=sAssetID, iotprops := st_IotProps);
					State.LastIndexSent := i;
					EXIT;
				END_IF
			END_IF
		END_IF
	END_FOR
ELSE
	RETURN;
END_IF

IF State.LastIndexSent = State.LastIndex AND State.bUpdate THEN
	State.bUpdate := FALSE;
	State.LastIndexSent := 0;
END_IF
END_METHOD

METHOD shutdown : BOOL
IF s_ShutdownFb = 'ERR' THEN
	w_shutdown := 0;
ELSE
	w_shutdown := 1;
END_IF

shutdown := s_ShutdownFb = 'OK';
END_METHOD

END_PROGRAM

// ---- POUs/MonitoringControl/ExternalControl/FB_ExternalController.TcPOU
FUNCTION_BLOCK FB_ExternalController
VAR_INPUT
	set				: ST_ExtController_Set;
END_VAR
VAR_OUTPUT
	get							: ST_ExtController_get;
END_VAR

VAR_IN_OUT CONSTANT
	{ attribute 'TcHmiSymbol.Hide' }
	monitor								: ST_System_Monitor;
END_VAR

//HMI controls to be overwritten from get if controller is allowed.
VAR_IN_OUT
	st_params							: ST_Extcontroller_params;
	controlvars							: ST_System_Control;
END_VAR

VAR
	ExternalControlMode			:	eExternalControlMode := eExternalControlMode.off;
	HeartBeatFault				:	Bool;
END_VAR

VAR
	Inputs						:	ST_PNInput;
	Outputs				AT %Q*	:	ST_PNOutput;
	
	PNInputs			AT %I*	:	ST_PNInput;
	MBInputs			AT %I*	:	ST_PNInput;
	MBInputsV2			AT %I*	:	ST_PNInput; //output can be mapped to the same struct as V1
	
	BindControlvars				: FB_BindControlvars;
	
	e_ID						: eObject_ID := eObject_ID.PNcontroller;
	
	fTrigTestScript				: F_Trig;
	emptyEventStruct			: ST_ExtController_Events;
	emptyTestStruct				: ST_PNTest;
	TestScript					: FB_ExtControllerTest;
	
	b_enableByteSwap			: BOOL;
END_VAR

VAR
	monitoringvalues			: REFERENCE TO ST_System_Monitor;
	
	fbJson         	: FB_JsonSaxWriter;
  	fbJsonDataType 	: FB_JsonReadWriteDataType;
  	sJsonDoc2       				: STRING(2000); 
	rtrig_SwitchToExtControl	:	r_trig;
	ManualAckState	:	BOOL;

	bTest:bool;
END_VAR


get.control.b_ActivateSettings := (ExternalControlMode = eExternalControlMode.AdvancedControl);

IF settings.Configuration.e_PNcouplerType <> ePNcouplerType.None  THEN
	CASE settings.Configuration.e_PNcouplerType OF
		ePNCouplertype.ModbusTCP:	 	Inputs := MBInputs;
		ePNCouplerType.ModbusTCPV2: 	Inputs := MBInputsV2;
		ePNCouplerType.Profinet:		Inputs := PNInputs;
	END_CASE
	
	CheckControlMode();
	
	IF CheckCouplerState() or bTest THEN //wait for coupler to be present
		IF (ExternalControlMode > eExternalControlMode.Readonly) AND NOT get.events.b_HeartbeatFault THEN
			get.e_ConnectionState := eConnectionState.authorized;
		ELSIF NOT get.events.b_HeartbeatFault THEN
			get.e_ConnectionState := eConnectionState.connected;
		ELSE
			get.e_ConnectionState := eConnectionState.disconnected;
		END_IF
	
		IF ExternalControlMode > eExternalControlMode.off THEN //only write outputs if monitoring is allowed
		
			//always check the heartbeat input, only process the events when Externalcontrolmode > readonly
			Outputs.General.ui_HeartBeatOut := wordEndian(HeartBeat(ui_HeartBeatInput := Inputs.General.ui_HeatBeat, b_heartbeatfault => HeartBeatFault));
			get.events.b_HeartbeatFault := SEL(ExternalControlMode > eExternalControlMode.Readonly, FALSE, HeartBeatFault);
			get.ui_Heartbeat := Inputs.general.ui_HeatBeat;
		
			MapGeneralData		(Monitor := monitor, Input := Inputs.General, 			Output := Outputs.General, 				events:= get.events	);
			MapBatteryData		(Monitor := monitor, Input := Inputs.Battery,			Output := Outputs.Battery			,	events:= get.events	);
			MapOutputField		(Monitor := monitor,									Output := Outputs.OutputField								);
			MapInputField		(Monitor := monitor, Input := Inputs.Inputfield, 		Output := Outputs.InputField		, 	events:= get.events	);
			MapPowerStack		(Monitor := monitor, Input := Inputs.Powerstack,	 	Output := Outputs.Powerstack		, 	events:= get.events	);
			MapPeakShaveBox		(Monitor := monitor, Input := Inputs.PSB, 				Output := Outputs.PSB				,	events:= get.events	);
			MapZPT				(Monitor := monitor,									Output := Outputs.ZPT										);
			MapGeneratorControl	(Monitor := monitor, Input := inputs.GenControl,		Output := Outputs.GenControl		,	events := get.events);
			MapInputGridControl	(Monitor := monitor, Input := inputs.InputGridControl,	Output := Outputs.InputGridControl	, 	events := get.events);	
			MapACDCCharger		(monitor := monitor, input := inputs.ACDCCharger, 		output := outputs.ACDCCharger		,	events := get.events);	
			
			IF ExternalControlMode > eExternalControlMode.Readonly THEN
				BindControlVars(AdvancedControl :=  ExternalControlMode = eExternalControlMode.AdvancedControl,
								SystemControlVars := controlvars, 
								ExtControlVars := get);
			END_IF
		END_IF
	
		rtrig_SwitchToExtControl(clk := monitor.controlfb.HardSettings.setup.e_ControlSource = eControlSources.ExternalController);	
		IF rtrig_SwitchToExtControl.q THEN
			get.control := controlvars.control;
			get.HardSettings := controlvars.HardSettings;
			get.Operation := controlvars.Operation;
			get.SoftSettings := controlvars.SoftSettings;
		END_IF
	END_IF
ELSE
	get.events.b_CouplerError := FALSE;
	get.events.b_HeartbeatFault := FALSE;
	ExternalControlMode := eExternalControlMode.off;
END_IF

		
SetJsonDoc(get.s_OutputJson);

METHOD CheckControlMode : BOOL
VAR_INPUT
	
END_VAR

IF monitor.controlfb.HardSettings.setup.e_ControlSource = eControlSources.ExternalController THEN
	IF get.b_AdvancedControl THEN
		ExternalControlMode := eExternalControlMode.AdvancedControl;
	ELSE
		ExternalControlMode := eExternalControlMode.BasicControl;
	END_IF
ELSIF st_params.b_MonitoringEnable THEN
	ExternalControlMode := eExternalControlMode.Readonly;
ELSE
	ExternalControlMode := eExternalControlMode.off;
END_IF
END_METHOD

METHOD CheckCouplerState : BOOL
VAR_INPUT

END_VAR
//TBD: Verder uitbereiden

IF Inputs.PNIOBoxState = 0 THEN // = No error
	CheckCouplerState := TRUE;
	get.events.b_CouplerError := FALSE;
ELSE
	CheckCouplerState := FALSE;
	get.events.b_CouplerError := TRUE;
//1 = Profinet device state machine is in boot mode
//2 = Device not found
//3 = The stationname is not unique
//4 = IP could not be set
//5 = IP conflict
//6 = DCP set was not successful
//7 = Watchdog error
//8 = Datahold error
//9 = RTC3: Sync mode could not be initiated
//10 = Profinet controller has a link error
//11 = The aliasname is not unique
//12 = The automatic name assignement isn't possible - wrong device type
//13 = IOC-AR is established but no application ready
//14 = IOC-AR is established but module difference
//15 = At least one InputCR is invalid, provider in stop or problemindicator is set
//16 = At least one OutputCR is invalid, provider in stop or problemindicator is set
//31 = Only for EtherCAT gateways: WC-State of cyclic EtherCAT frame is 1
END_IF
END_METHOD

METHOD DwordEndian : DWORD
VAR_INPUT
	IN		: DWORD;
END_VAR
IF st_params.b_BigEndian THEN
	DwordEndian := HOST_TO_BE32(IN);
ELSE
	DwordEndian := IN;
END_IF
END_METHOD

METHOD DwordToReal : REAL
VAR_INPUT
	InputVar			:	DWORD;
	b_InputSigned		:	BOOL;
	Stepsize			:	WORD;
end_var
DwordToReal := 1;

IF b_inputSigned AND InputVar.31 THEN
	DwordToReal := -1;
	InputVar.31 := FALSE;
END_IF

DwordToReal := DwordToReal * DWORD_TO_REAL(InputVar)/Stepsize;
END_METHOD

METHOD GenGridControllerStateMachine : BOOL
VAR_INPUT
END_VAR

VAR_INST
	State		:	UINT;
	rTrig_Ack	:	R_trig;
	test		:	BOOL;
	AckDelay	:	Ton := (pt := T#1S200ms);
END_VAR
get.Operation.system.b_GenGridModeTrans := FALSE;
rTrig_Ack(clk := ManualAckState);
AckDelay();
//get.Operation.system.b_GenGridModeTrans := Ackdelay.q;
AckDelay.IN := FALSE;

CASE monitor.system.GenGridController.e_BreakerMode OF
	eBreakerOperationMode.none:
		AckDelay.IN := FALSE;
		//IF monitor.system.GenGridController.b_ModeTransActive THEN
		//	get.Operation.system.b_GenGridModeTrans := TRUE;
		//END_IF
		
	eBreakerOperationMode.GridFeedthrough:
		IF get.SoftSettings.setup.e_AcInputType = eAcInputType.Grid THEN
			IF get.SoftSettings.inputgrid.breaker.AutoConnect THEN	//connect if requested, otherwise hold here
				IF monitor.system.GenGridController.b_ModeTransActive THEN
					get.Operation.system.b_GenGridModeTrans := TRUE;
				END_IF
			ELSE 
				IF monitor.system.GenGridController.e_state = eGenGridSTate.Running then
					get.Operation.system.b_GenGridModeTrans := TRUE;
				END_IF
			END_IF		
		END_IF	
		IF get.SoftSettings.setup.e_AcInputType = eAcInputType.None THEN //transitioning to none
			IF (NOT get.SoftSettings.inputgrid.breaker.AutoConnect OR rTrig_ack.q) AND monitor.ACswitchgear.b_InputContactorfb THEN
				get.Operation.system.b_GenGridModeTrans := TRUE;
			elsIF NOT monitor.ACswitchgear.b_InputContactorfb AND monitor.system.GenGridController.b_ModeTransActive THEN
				AckDelay.in := TRUE;
				get.Operation.system.b_GenGridModeTrans := AckDelay.q;
			END_IF//get.Operation.system.b_GenGridModeTrans := true;//rTrig_Ack.q;
		END_IF
	
	eBreakerOperationMode.GenIso: //eBreakerOperationMode.GenDroop, 
		IF get.SoftSettings.setup.e_AcInputType = eAcInputType.None THEN //transitioning to none	
			IF monitor.ACswitchgear.b_InputContactorfb THEN
				get.Operation.system.b_GenGridModeTrans := rTrig_Ack.Q;
			ELSIF monitor.system.GenGridController.b_ModeTransActive THEN
				AckDelay.in := TRUE;
				get.Operation.system.b_GenGridModeTrans := AckDelay.q;
			END_IF//get.Operation.system.b_GenGridModeTrans := true;//rTrig_Ack.q;
		END_IF
		
	eBreakerOperationMode.GenFix:
		IF get.SoftSettings.setup.e_AcInputType = eAcInputType.None THEN //transitioning to none	
			IF monitor.ACswitchgear.b_InputContactorfb THEN
				IF NOT (monitor.system.GenGridController.e_state = eGenGridState.Cooldown OR 
						monitor.system.GenGridController.e_state = eGenGridState.Running OR
						monitor.system.GenGridController.e_state = eGenGridState.Warmup) THEN
					get.Operation.system.b_GenGridModeTrans := true;
				ELSE	
					get.Operation.system.b_GenGridModeTrans := rTrig_Ack.Q;
				end_if
			ELSIF monitor.system.GenGridController.b_ModeTransActive THEN
				AckDelay.in := TRUE;
				get.Operation.system.b_GenGridModeTrans := AckDelay.q;
			END_IF//get.Operation.system.b_GenGridModeTrans := true;//rTrig_Ack.q;
		END_IF
END_CASE



//get.SoftSettings.inputgenset.b_AutoStartStop := (inputs.General.SecondaryDigOutState = 1 OR inputs.GenControl.ui_StartStopControl = 1);

//IF (inputs.General.SecondaryDigOutState = 2 OR inputs.GenControl.ui_StartStopControl = 2) THEN
//	IF monitor.system.GenGridController.e_RunCondition <> eruncondition.ManuallyStarted THEN
//		get.Operation.Genset.b_manualStart := NOT get.Operation.Genset.b_manualStart;
//	END_IF
//ELSIF (inputs.General.SecondaryDigOutState <> 2 AND inputs.GenControl.ui_StartStopControl <> 2) AND monitor.system.GenGridController.e_RunCondition = eruncondition.ManuallyStarted THEN
//		get.Operation.Genset.b_manualStart := NOT get.Operation.Genset.b_manualStart;
//END_IF

//CASE State OF
//	0: //none
//		Ackdelay.IN := FALSE;
//		CASE get.SoftSettings.setup.e_AcInputType OF
//			eAcInputType.Grid: //transitioning to grid
//				State := 1; //switch to gridInit
//			eAcInputType.Genset: //transitioning to grid
//				State := 3; //switch to gridInit
//		END_CASE
//	1: //gridInit
//		CASE get.SoftSettings.setup.e_AcInputType OF
//			eAcInputType.Grid: //transitioning to grid
//				IF get.SoftSettings.inputgrid.breaker.AutoConnect THEN	//connect if requested, otherwise hold here
//					IF monitor.system.GenGridController.b_ModeTransActive THEN
//						get.Operation.system.b_GenGridModeTrans := TRUE;
//					END_IF
//					State := 2; //SwitchToGridActive	
//				END_IF
				
//			eACInputType.None: //transitioning to none
//				AckDelay.IN := (NOT monitor.system.GenGridController.b_active) AND monitor.system.GenGridController.e_State = eGenGridState.Waiting_Mode_Reconnect;
//				IF AckDelay.q THEN
//					IF monitor.system.GenGridController.b_ModeTransActive THEN
//						get.Operation.system.b_GenGridModeTrans := TRUE;
//					END_IF//get.Operation.system.b_GenGridModeTrans := true;//rTrig_Ack.q;
//				END_IF
				
//				IF monitor.system.GenGridController.e_State = eGenGridState.Init THEN
//					get.Operation.system.b_GenGridModeTrans := FALSE;
//					State := 0;
//				END_IF;
//		END_CASE
		
//	2: //GridModeActive
		
//		//get.Operation.system
//		IF NOT get.SoftSettings.inputgrid.breaker.AutoConnect or rTrig_Ack.q THEN
//			//IF monitor.system.GenGridController.e_state = eGenGridSTate.Running OR 
//				//monitor.system.GenGridController.e_state = eGenGridSTate.Synchronization THEN
//			//	 Ackdelay.IN := TRUE;
//			//ELSE
//			//	Ackdelay.IN := FALSE;
//				get.Operation.system.b_GenGridModeTrans := TRUE;
//				State := 1;
//			//END_IF
//		ELSE
//			IF NOT monitor.ACswitchgear.b_InputContactorfb THEN
//				State := 1;
//			END_IF
//		END_IF
		
//	3:	//GenMode
////		CASE get.SoftSettings.setup.e_AcInputType OF				
////			eACInputType.None: //transitioning to none
////				AckDelay.IN := (NOT monitor.system.GenGridController.b_active) AND monitor.system.GenGridController.e_State = eGenGridState.Waiting_Mode_Reconnect;
////				IF AckDelay.q THEN
////					IF monitor.system.GenGridController.b_ModeTransActive THEN
////						get.Operation.system.b_GenGridModeTrans := TRUE;
////					END_IF//get.Operation.system.b_GenGridModeTrans := true;//rTrig_Ack.q;
////				END_IF
				
////				IF monitor.system.GenGridController.e_State = eGenGridState.Init THEN
////					get.Operation.system.b_GenGridModeTrans := FALSE;
////					State := 0;
////				END_IF;
////		END_CASE

//		//IF rTrig_Ack.Q THEN
//		//	get.Operation.system.b_GenGridModeTrans := TRUE; 
//		//	State := 1;
//		//END_IF
//END_CASE

////CASE WordEndian(Input.InputConnectionType) OF
////		//0:	remain
////		1:	get.SoftSettings.setup.e_AcInputType := eAcInputType.None; 
////		2:	get.SoftSettings.setup.e_AcInputType := eAcInputType.Grid;
////		3:	get.SoftSettings.setup.e_AcInputType := eAcInputType.Genset; 
////	END_CASE
END_METHOD

METHOD GetDiagnostics : BOOL
VAR_IN_OUT
	AddError		: ARRAY [*] OF FB_AddErrorST;
	a_ActiveEvents	: ARRAY [*] OF ST_ErrorStruct;
	w_Index			: WORD;
END_VAR

VAR_OUTPUT
	b_errorActive	: BOOL;
	b_warningActive	: BOOL;
END_VAR

VAR_INST
	by_errCt	: BYTE;
	by_warnCt	: BYTE;
END_VAR
	(*Watchdog fault*)	AddError[w_Index](
			b_ErrorTrig			:= Get.Events.b_HeartbeatFault,
			out_ST_Error			:= a_ActiveEvents[w_Index],
			w_ErrorID					:= 1,
			e_ObjectID				:= e_id,
			s_Message				:= 'watchdog fault',
			e_sev					:= eSeverity.warning,	
			b_AutoClear			:= TRUE,
			e_ErrAckAccess		:= eErrAckAccess.Operator,
			);
		w_Index := w_Index +1;
		
	(*Coupler fault*)	AddError[w_Index](
			b_ErrorTrig			:= Get.events.b_CouplerError,
			out_ST_Error			:= a_ActiveEvents[w_Index],
			w_ErrorID				:= 2,
			e_ObjectID				:= e_id,
			s_Message				:= concat('External control interface error: ', TO_STRING(Inputs.PNIOBoxState)),
			t_TriggerTime			:=	T#30S,
			e_sev					:= eSeverity.info,	
			b_AutoClear				:= TRUE,
			e_ErrAckAccess			:= eErrAckAccess.Operator,
			);
		w_Index := w_Index +1;
END_METHOD

METHOD HeartBeat : UINT
VAR_INPUT
	ui_HeartBeatInput		:	UINT	:=	0;
END_VAR

VAR_OUTPUT
	b_HeartBeatFault		:	BOOL;
END_VAR

VAR_INST
	ui_HeartBeatOutput			:	UINT ; 
	HeartBeatOutputIncTimer		:	TON		:=	(PT := T#500MS);
	HeartBeatInputCheckTimer	:	TON		:=	(PT := T#1S);
	ui_StoredInputValue			:	UINT	:= 	0;

END_VAR

//output value increments every second. Remote party should check if this happens
HeartBeatOutputIncTimer (in := NOT HeartBeatOutputIncTimer.Q);
IF HeartBeatOutputIncTimer.Q THEN
	ui_HeartBeatOutput := ui_HeartBeatOutput +1;
END_IF

//Input value has to change every second as well.
//if stored and Current values are equal, start counting.
HeartBeatInputCheckTimer(in:= (ui_StoredInputValue = ui_HeartBeatInput), PT := TO_TIME(st_params.w_CommTimeOut));
ui_StoredInputValue := ui_HeartBeatInput;
b_heartBeatFault := HeartBeatInputCheckTimer.Q;

Heartbeat := ui_HeartBeatOutput;
END_METHOD

METHOD IntToReal : BOOL
VAR_INPUT
	in			:	INT;
	Scale		:	UINT := 10;
	LimitLow	: 	REAL := -3.402823E+38;
	LimitHigh	:  	REAL := 3.402823E+38; 
	IgnoreZero	:	BOOL := FALSE;
END_VAR

VAR_OUTPUT
	OutofRange	: BOOL;
END_VAR

VAR
	r_value			: 	REAL;
	test			:	INT;
	test2			:	real;
END_VAR

VAR_IN_OUT
	Out	:	REAL;
END_VAR

IF (NOT IgnoreZero) OR (in <> 0) THEN
	test := WordEndian(in);
	test2 := INT_TO_REAL(test);
	r_value	 := test2/Scale;
	
	OutofRange := ValueOutOfRange(r_value, LimitLow, LimitHigh);
	Out := LIMIT(LimitLow, r_value, LimitHigh);
END_IF
END_METHOD

METHOD MapACDCCharger : BOOL
VAR_IN_OUT CONSTANT
	monitor								: ST_System_Monitor;
END_VAR

VAR_IN_OUT
	events	: 	ST_ExtController_Events;
	Input	:	st_PNInput_ACDCCharger;
	Output	:	st_PNOutput_ACDCCharger;
END_VAR

VAR_INST
	rtrig_openInputBreaker	:	r_trig;
	Rtrig_BreakerToAuto		:	r_trig;
	ftrig_ackDone			:	f_trig;
END_VAR



IF NOT settings.MachineParams.ACDCCharger.b_ACDCChargerFitted THEN
	output.w_Status := 0;
ELSE
	output.w_Status.15	:=	settings.MachineParams.ACDCCharger.b_ACDCChargerFitted;
	output.w_Status.10	:=	monitor.AcDcCharger.Events.b_BatteryLimitDeratingActive;
	output.w_Status.9	:=	monitor.AcDcCharger.Events.b_ACUnderVoltageDeratingActive;
	output.w_Status.8	:=	monitor.AcDcCharger.Events.b_TemperatureDeratingActive;
	
	output.w_Status.1	:=	monitor.AcDcCharger.r_DcVoltage > 500;
	output.w_Status.0	:=	monitor.AcDcCharger.ar_ACvoltage[phases.AVG] > 200;
	output.w_Status := wordEndian(output.w_Status);
	
	
	//Fill output data
	Output.w_Warnings.3	:=	monitor.AcDcCharger.ar_ACvoltage[phases.AVG] > 430;
	Output.w_Warnings.2	:=	monitor.AcDcCharger.e_SystemStatus = eACDCChargerState.running AND
							monitor.AcDcCharger.ar_ACvoltage[phases.AVG] < 370;
	Output.w_Warnings.1	:=	monitor.AcDcCharger.Events.b_TemperatureDeratingActive;
	Output.w_Warnings.0	:=	FALSE;//monitor.AcDcCharger.Events.b_CommunicationFault
	Output.w_Warnings	:=  WordEndian(Output.w_Warnings);
	
	
	Output.w_Faults.7	:=	FALSE;//monitor.AcDcCharger.Events.DCOverVoltageFault;
	Output.w_Faults.6	:=	FALSE;//monitor.AcDcCharger.Events.DCUnderVoltageFault;
	Output.w_Faults.5	:=  FALSE;//monitor.AcDcCharger.Events.DCOverVoltageFault;
	Output.w_Faults.4	:=  monitor.AcDcCharger.Events.B_ACPhaselossFault;
	Output.w_Faults.3	:=  monitor.AcDcCharger.Events.B_ACOvervoltage;
	Output.w_Faults.2	:=	monitor.AcDcCharger.Events.B_ACUndervoltage;
	Output.w_Faults.1	:=	FALSE; //overtemperature fault
	Output.w_Faults.0	:=	monitor.AcDcCharger.Events.b_CommunicationFault OR 
							monitor.AcDcCharger.Events.b_BuscouplerNotFound;
	Output.w_Faults		:= 	WordEndian(Output.w_Faults);
	
	
	Output.ui_ChargerStatus := WordEndian(monitor.AcDcCharger.e_SystemStatus);
	
	output.TotalChargerPower := WordEndian(REAL_TO_UINT(monitor.AcDcCharger.by_NoModulesInstalled * 300));
	output.AvailableChargePower := WordEndian(REAL_TO_UINT(monitor.AcDcCharger.r_AvailablePower * 10));
	output.ActivePower	:=	WordEndian(REAL_TO_UINT(monitor.AcDcCharger.ACmeasurements.ar_ActivePower[0]*10));	
	output.Frequency 	:= wordendian(0);
	output.VoltageAB	:=	wordendian(REAL_TO_UINT(monitor.AcDcCharger.ar_ACvoltage[1]*10));
	output.VoltageBC	:=	wordendian(REAL_TO_UINT(monitor.AcDcCharger.ar_ACvoltage[2]*10));	
	output.VoltageCA	:=	wordendian(REAL_TO_UINT(monitor.AcDcCharger.ar_ACvoltage[3]*10));
	
	output.CurrentL1	:= wordendian(REAL_TO_UINT(monitor.acDcCharger.ACmeasurements.ar_Current[1]*10));
	output.CurrentL2	:= wordendian(REAL_TO_UINT(monitor.acDcCharger.ACmeasurements.ar_Current[2]*10));
	output.currentL3	:= wordendian(REAL_TO_UINT(monitor.acDcCharger.ACmeasurements.ar_Current[3]*10));
	
	output.ui_ACCurrentLimitAct := wordendian(REAL_TO_UINT(get.softsettings.ACDCcharger.r_CurrentSetpoint*10));
	output.ui_PSetAct 			:=	wordendian(REAL_TO_UINT(get.SoftSettings.ACDCcharger.r_PowerSetpoint*10));
	output.ui_SocLimitAct		:=	wordendian(REAL_TO_UINT(get.SoftSettings.ACDCcharger.r_SocTarget*10)); 
	output.ui_MinGridVoltageAct	:=	wordendian(REAL_TO_UINT(get.SoftSettings.ACDCcharger.r_MinACVoltage*10));
	
	IF (NOT events.b_HeartbeatFault) AND ExternalControlMode > eExternalControlMode.BasicControl AND monitor.system.GenGridController.e_BreakerMode = eBreakerOperationMode.GridFeedthrough THEN
		input.w_Control := wordEndian(input.w_Control);
		get.SoftSettings.ACDCcharger.b_Enable := input.w_Control.0;
		get.SoftSettings.ACDCcharger.e_ControlType := ePowerControltype.Both;
		
		UIntToReal(	in			:= Input.ui_ACCurrentlimit, 
					scale 		:= 10, 
					limitlow	:= 0,
					limithigh	:= 100,//get.HardSettings.inputgrid.r_FeedInCurrentLimitHard,
					OutOfRange 	=>	,
					IgnoreZero 	:= FALSE,
					Out 		:= get.SoftSettings.ACDCcharger.r_CurrentSetpoint);
		
		UIntToReal(	in			:= Input.UI_Pset, 
					scale 		:= 10, 
					limitlow	:= 0,
					limithigh	:= monitor.AcDcCharger.by_NoModulesInstalled*30,
					OutOfRange 	=>	,
					IgnoreZero 	:= FALSE,
					Out 		:= get.SoftSettings.ACDCcharger.r_PowerSetpoint);
	
		UIntToReal(	in			:= Input.ui_SocMaxLimit, 
					scale 		:= 10, 
					limitlow	:= 0,
					limithigh	:= 100,//get.HardSettings inputgrid.r_SupplyCurrentLimitHard,
					OutOfRange 	=>	,
					IgnoreZero 	:= TRUE,
					Out 		:= get.SoftSettings.ACDCcharger.r_SocTarget);
	
		UIntToReal(	in			:= Input.ui_MinGridVoltage, 
					scale 		:= 10, 
					limitlow	:= 360,
					limithigh	:= 440,//get.HardSettings inputgrid.r_SupplyCurrentLimitHard,
					OutOfRange 	=>	,
					IgnoreZero 	:= TRUE,
					Out 		:= get.SoftSettings.ACDCcharger.r_MinACVoltage);

	ELSE
		get.SoftSettings.ACDCcharger.r_PowerSetpoint := 0;
	END_IF
END_IF
END_METHOD

METHOD MapBatteryData : BOOL
VAR_IN_OUT CONSTANT
	monitor								: ST_System_Monitor;
END_VAR

VAR_IN_OUT
	events	: 	ST_ExtController_Events;
	Input	:	ST_PNInput_Battery;
	Output	:	ST_PNOutput_Battery;

END_VAR

Output.ui_Status := WordEndian(Monitor.battery.BatteryInfo.e_BMS_Status);

Output.w_Warnings.0 := Monitor.battery.events.b_OVER_TEMP_WARNING;	
Output.w_Warnings.1 := Monitor.battery.events.b_UNDER_TEMP_WARNING;			
Output.w_Warnings.2 := Monitor.battery.events.b_OVER_CHARGE_CURRENT_WARNING;	
Output.w_Warnings.3 := Monitor.battery.events.b_OVER_DISCHARGE_CURRENT_WARNING;
Output.w_Warnings.4 := Monitor.battery.events.b_OVER_VOLT_WARNING;		
Output.w_Warnings.5 := Monitor.battery.events.b_UNDER_VOLT_WARNING;		
Output.w_Warnings.6 := Monitor.battery.events.b_UNDER_SOC_MIN_WARNING;		
Output.w_Warnings.7 := Monitor.battery.events.b_OVER_SOC_MAX_WARNING;			
Output.w_Warnings.8 := Monitor.battery.events.b_VOLTAGE_IMBALANCE_WARNING;
Output.w_Warnings.9 := Monitor.battery.events.b_TEMPERATURE_IMBALANCE_WARNING;
Output.w_Warnings.10 := Monitor.battery.events.b_CURRENT_IMBALANCE_WARNING;
Output.w_Warnings.11 := Monitor.battery.events.b_OTHER_WARNING;	
Output.w_Warnings.12 := Monitor.battery.events.b_CONFIGURATION_WARNING;
Output.w_Warnings := WordEndian(Output.w_warnings);

Output.w_Faults.0 := Monitor.battery.Events.b_COMMUNICATION_ERROR;			
Output.w_Faults.1 := Monitor.battery.events.b_OVER_TEMP_ALARM;					
Output.w_Faults.2 := Monitor.battery.events.b_UNDER_TEMP_ALARM;			
Output.w_Faults.3 := Monitor.battery.events.b_OVER_CHARGE_CURRENT_ALARM;		
Output.w_Faults.4 := Monitor.battery.events.b_OVER_DISCHARGE_CURRENT_ALARM;	
Output.w_Faults.5 := Monitor.battery.events.b_OVER_VOLT_ALARM;						
Output.w_Faults.6 := Monitor.battery.events.b_UNDER_VOLT_ALARM;					
Output.w_Faults.7 := Monitor.battery.events.b_UNDER_SOC_MIN_ALARM;				
Output.w_Faults.8 := Monitor.battery.events.b_OVER_SOC_MAX_ALARM;				
Output.w_Faults.9 := Monitor.battery.events.b_TEMPERATURE_IMBALANCE_ALARM;	
Output.w_Faults.10 := Monitor.battery.events.b_CONTACTOR_ERROR;				
Output.w_Faults.11 := Monitor.battery.events.b_FAN_ERROR;						
Output.w_Faults.12 := Monitor.battery.events.b_GROUND_FAULT;					
Output.w_Faults.13 := Monitor.battery.events.b_OPEN_DOOR_ERROR;					
Output.w_Faults.14 := Monitor.battery.events.b_OTHER_ALARM;								
Output.w_Faults.15 := Monitor.battery.events.b_CONFIGURATION_ALARM;	
Output.w_Faults := WordEndian(Output.w_Faults);		
			
Output.ui_SOC 							:= RealToUint(	In	:=	monitor.battery.BatteryInfo.r_SOCScaled, 	Scale	:=	10);
Output.ui_SOH 							:= RealToUint(	In	:=	monitor.battery.BatteryInfo.r_SOH, 	Scale	:=	10);
Output.ui_DClinkVoltage 				:= RealToUint(	In	:=	monitor.battery.BatteryInfo.r_SystemVoltage, Scale	:=	10);				
Output.i_DClinkCurrent 					:= RealToint (	In	:=	monitor.battery.BatteryInfo.r_SystemCurrent, Scale	:=	10);
Output.ui_MaxAllowedDischargeCurrent 	:= RealToUint (	In	:=	monitor.battery.BatteryInfo.r_MaxDischargeCurrentAllowed, Scale	:=	10); 	
Output.ui_MaxAllowedChargeCurrent 		:= RealToUint (	In	:=	-monitor.battery.BatteryInfo.r_MaxchargeCurrentAllowed,	Scale	:=	10); 		
Output.i_MinCellTemperature 			:= RealToint (	In	:=	monitor.battery.BatteryInfo.ar_CellTemperature[0] , Scale	:=	10); 	
Output.i_MaxCellTemperature				:= RealToint (	In	:=	monitor.battery.BatteryInfo.ar_CellTemperature[2], Scale	:=	10); 										                                               
Output.ui_RemainingChargeEnergy 		:= RealToUint(	In	:=	monitor.battery.BatteryInfo.r_RemainingChargeEnergy, Scale	:=	10);
Output.ui_RemainingDischargeEnergy 		:= RealToUint(	In	:=	monitor.battery.BatteryInfo.r_RemainingDischargeEnergy, Scale	:=	10);
Output.ui_CycleCount					:= WordEndian(monitor.battery.BatteryInfo.ui_CycleCount);

//Read regularinputs if allowed
IF (NOT events.b_HeartbeatFault) AND ExternalControlMode > eExternalControlMode.BasicControl THEN
	Input.w_Control := WordEndian(input.W_Control);
	get.Operation.BMS.b_ManualStartHVDC := Input.W_Control.0;
		
	UintToReal(	in			:= 	Input.ui_SocMinLimit, 
				scale 		:= 	10, 
				limitlow	:=	0, 
				limithigh	:=	90, 
				OutOfRange 	=>	events.b_SoCLowLimitOutOfRange,
				IgnoreZero 	:= 	FALSE,
				Out 		:= 	get.softsettings.system.r_SocMin);

	UintToReal(	in			:= 	Input.ui_SocMaxLimit, 
				scale 		:= 	10, 
				limitlow	:=	10, 
				limithigh	:=	100, 
				OutOfRange 	=>	events.b_SoCHighLimitOutOfRange,
				IgnoreZero 	:= 	TRUE,
				Out 		:= 	get.softsettings.system.r_SocMax);	
END_IF
END_METHOD

METHOD MapGeneralData : BOOL
VAR_IN_OUT CONSTANT
	monitor								: ST_System_Monitor;
END_VAR

VAR_IN_OUT
	events	: 	ST_ExtController_Events;
	Input	:	ST_PNInput_general;
	Output	:	ST_PNOutput_general;
END_VAR

VAR
	SWVersion	:	uSWversion;
END_VAR

VAR_INST
	b_PENMissingTrip	:	BOOL;
	rtrig_disconnectNetcontactor	:	r_trig;
	ftrig_disconnectNetcontactor	:	f_trig;
	
	rtrig_GridToNone	: r_trig;
END_VAR
//First check heartbeat status
events.b_GridModeValueOutOfRange := FALSE;
events.b_PowermodeValueOutOfRange:= FALSE;

Output.ui_SystemState		:=	WordEndian(TO_UINT(Monitor.system.e_State));
	
Output.w_SystemStatus.0		:= 	Monitor.protections.Insulation.b_Enabled;
Output.w_SystemStatus.1		:= 	ExternalControlMode > eExternalControlMode.Readonly;
Output.w_SystemStatus.2		:=	monitor.protections.FireDetection.b_FireAlarm AND NOT monitor.protections.FireDetection.Events.AlarmMuted;
Output.w_SystemStatus.3		:=	monitor.HartingIO.b_DigitalInput1Active;
output.w_SystemStatus.4		:=	monitor.HartingIO.b_DigitalInput2Active;
Output.w_SystemStatus.8		:=	monitor.protections.Insulation.e_EarthingSystemDetected = eEarthingSystems.TN;//Monitor.system.e_EarthingSystem = eEarthingSystems.TN;
Output.w_SystemStatus.9		:=	monitor.protections.Insulation.e_EarthingSystemDetected = eEarthingSystems.IT;//Monitor.system.e_EarthingSystem = eEarthingSystems.IT;
Output.w_SystemStatus		:= 	WordEndian(Output.w_SystemStatus);
	
Output.w_SystemWarnings.0	:=	Monitor.protections.FireDetection.CODetectors.State = eCOAlarmStatus.WarningLevel1;
Output.w_SystemWarnings.1	:=	Monitor.protections.FireDetection.CODetectors.State = eCOAlarmStatus.WarningLevel2;
Output.w_SystemWarnings.2	:=	Monitor.protections.Insulation.b_Warning;
Output.w_SystemWarnings.3	:=	Monitor.protections.MRCDB.b_prewarning;
Output.w_SystemWarnings.8	:=	Monitor.protections.FireDetection.Events.SmokeDetFault;
Output.w_SystemWarnings.9	:=	Monitor.protections.FireDetection.Events.CODetFault;
Output.w_SystemWarnings.10	:=	NOT Monitor.protections.Surge.b_Type12_OK;
Output.w_SystemWarnings.11	:=	NOT Monitor.protections.Surge.b_Type3_OK;
Output.w_SystemWarnings.12	:=	Monitor.enclosure.doors.b_ControlPanelDoorOpen;
Output.w_SystemWarnings.13	:=	Monitor.enclosure.doors.b_ClientpanelDoorOpen;
Output.w_SystemWarnings 	:= 	WordEndian(Output.w_SystemWarnings);

Output.w_SystemFaults.0		:=	Monitor.protections.FireDetection.Events.SmokeDetAlarm;
Output.w_SystemFaults.1		:=	Monitor.protections.FireDetection.Events.CODetAlarm;
Output.w_SystemFaults.2		:=	NOT Monitor.safety.b_InsulationMonitorOK;
Output.w_SystemFaults.3		:=	NOT Monitor.safety.b_MRCDBOK;
Output.w_SystemFaults.4		:=	NOT Monitor.safety.b_EstopChannelAOK OR NOT Monitor.safety.b_EstopChannelBOK;
Output.w_SystemFaults.5		:=	NOT Monitor.safety.b_SafetyOK;

Output.w_SystemFaults.6		:=	monitor.protections.Insulation.b_EarthingSystemMismatch OR 
								monitor.protections.Insulation.b_NoEarthingSystemSet OR 
								monitor.protections.Insulation.b_PENlinkOperatedFault OR 
								b_PENMissingTrip;
Output.w_SystemFaults.8		:=	NOT Monitor.safety.b_InverterDoorOK;
Output.w_SystemFaults 		:= 	WordEndian(Output.w_SystemFaults);								

Output.w_CoolingSystemStatus.0	:=	Monitor.Cooling.CoolingSystemState = eCoolingSystemState.OFF;
Output.w_CoolingSystemStatus.1	:=	Monitor.Cooling.CoolingSystemState= eCoolingSystemState.Circulating;
Output.w_CoolingSystemStatus.8	:=	Monitor.Cooling.HeatPumpStatus = eHeatPumpState.Active_Cooling;
Output.w_CoolingSystemStatus.9	:=	Monitor.Cooling.HeatPumpStatus = eHeatPumpState.Active_Heating;
Output.w_CoolingSystemStatus 	:= WordEndian(Output.w_CoolingSystemStatus);

Output.w_CoolingSystemWarnings.0	:=	Monitor.Cooling.Events.b_CoolantTempHigh;
Output.w_CoolingSystemWarnings.1	:=	Monitor.Cooling.Events.b_CoolantTempLow;
// Output.w_CoolingSystemWarnings.2	:=	Monitor.Cooling.Events.b_CoolingLoopIdlePressureWarning;
// Output.w_CoolingSystemWarnings.3	:=	Monitor.Cooling.Events.b_HeatPumpError;
// Output.w_CoolingSystemWarnings.4	:=	Monitor.Cooling.Events.b_FancoilLoopValveStuck;
Output.w_CoolingSystemWarnings.5	:=	Monitor.Cooling.Events.b_CoolingSystemFuseFailure;
Output.w_CoolingSystemWarnings		:= WordEndian(Output.w_CoolingSystemWarnings);
	
// Output.w_CoolingSystemFaults.1	:=	Monitor.Cooling.Events.b_BattLoopValveStuck OR Monitor.Cooling.Events.b_InverterLoopValveStuck;
// Output.w_CoolingSystemFaults.2	:=	Monitor.Cooling.Events.b_CoolingLoopIdlePressureError;									
//Output.w_CoolingSystemFaults.3	:=	Monitor.Cooling.Events.b_HeatpumpError;
Output.w_CoolingSystemFaults	:= 	WordEndian(Output.w_CoolingSystemFaults);
		
Output.w_InternalSupplyStatus.0	:=	Monitor.internalpsu.b_24VdcAvailable;
Output.w_InternalSupplyStatus.1	:=	Monitor.internalpsu.b_400VACAvailable;
Output.w_InternalSupplyStatus.2	:=	Monitor.internalpsu.b_HVDCAvailable;
Output.w_InternalSupplyStatus.3	:=	Monitor.internalpsu.UPS.b_SystemOnBattery;
Output.w_InternalSupplyStatus.4	:=	Monitor.internalpsu.UPS.b_ChargerActive;
Output.w_InternalSupplyStatus	:= 	WordEndian(Output.w_InternalSupplyStatus);

Output.w_InternalSupplyWarnings.0 := Monitor.internalpsu.UPS.Events.b_BatteryLowWarning;
//Output.w_InternalSupplyWarnings.1 := Monitor.internalpsu.Events.b_CEEInputFuseTripped;
Output.w_InternalSupplyWarnings.2 := Monitor.internalpsu.Events.b_ACPSUFault;
Output.w_InternalSupplyWarnings.3 := Monitor.internalpsu.Events.b_DCPSUFault;
Output.w_InternalSupplyWarnings	:= 	WordEndian(Output.w_InternalSupplyWarnings);

Output.w_InternalSupplyFaults.0 :=	Monitor.internalpsu.UPS.Events.b_BatteryLowError;
Output.w_InternalSupplyFaults.1 :=	monitor.internalpsu.Events.b_ACPSUFault AND monitor.internalpsu.Events.b_DCPSUFault;
Output.w_InternalSupplyFaults.3 :=	Monitor.internalpsu.Events.b_GridInputFuseTripped;
Output.w_InternalSupplyFaults	:= 	WordEndian(Output.w_InternalSupplyFaults);

IF Monitor.powerstack.e_InverterMode = eInverterModes.Island THEN
	Output.ui_Gridmode				:= 	WordEndian(TO_UINT(eGridmode.forming)+1);
	Output.ui_GridFormingSubMode	:= 	WordEndian(TO_UINT(eUgridPowermode.None)+1);
ELSIF Monitor.powerstack.e_InverterMode = eInverterModes.Afe THEN
	Output.ui_Gridmode				:= 	WordEndian(TO_UINT(eGridmode.following)+1);
	Output.ui_GridFormingSubMode	:= 	WordEndian(TO_UINT(eUgridPowermode.auto)+1);
ELSE
	Output.ui_Gridmode				:= 	WordEndian(TO_UINT(eGridmode.forming)+1);
	Output.ui_GridFormingSubMode	:= 	WordEndian(TO_UINT(monitor.system.e_UgridPowermode)+1);
END_IF
	
output.udi_SerialNumber			:=	DwordEndian(STRING_TO_UDINT(settings.Properties.s_SerialNumber));

SWVersion.a4byte_SWVer[3] := settings.Properties.by_SWverMajor;
SWVersion.a4byte_SWVer[2] := settings.Properties.by_SWverMinor;
SWVersion.a4byte_SWVer[1] := settings.Properties.by_SWverPatch;
SWVersion.a4byte_SWVer[0] := settings.Properties.by_SWverBuild;

//To do: Parse version number from config string
output.dw_SWVersion :=	DWordEndian(SWVersion.UD_SWVer);
	

//Read basic inputs if heartbeat is healthy
IF (NOT events.b_HeartbeatFault) THEN
	Input.W_Control := WordEndian(input.W_Control);
	//ControlVars.control.b_start := Input.W_Control.0;
	get.control.b_start 							:= Input.W_Control.0;
	get.control.b_shutdown 							:= Input.W_Control.2;
	controlvars.control.b_SystemShutdown			:=	Input.W_Control.3;
	//get.control.b_SystemShutdown					:= Input.W_Control.3;
	get.control.b_Reset 							:= Input.W_Control.4;
	get.control.b_EMstop 							:= Input.W_Control.5;
	get.SoftSettings.system.b_AutomaticSwitching 	:= Input.W_Control.6;
	get.SoftSettings.system.b_EnableTransportMode	:= Input.W_Control.7;
	get.b_AdvancedControl							:= Input.W_Control.9;

	//read other inputs if externalcontrol is active
	IF ExternalControlMode = eExternalControlMode.AdvancedControl THEN
		CASE WordEndian(Input.ui_GridMode) OF
			//0: 	remain
			1:	get.softsettings.setup.e_Gridmode := eGridMode.auto;
			2:	get.softsettings.setup.e_Gridmode := eGridMode.following;
			3:	get.softsettings.setup.e_Gridmode := eGridMode.forming;
		END_CASE
		
		CASE WordEndian(Input.ui_GridFormingSubMode) OF
			//0: 	remain
			1:	get.softsettings.system.e_UgridPowerMode := eUgridPowermode.auto;
			2:	get.softsettings.system.e_UgridPowerMode := eUgridPowermode.DroopZeroStart;
			3:	get.softsettings.system.e_UgridPowerMode := eUgridPowermode.Droop;
			4:	get.softsettings.system.e_UgridPowerMode := eUgridPowermode.Isochronous;
			5:	get.SoftSettings.system.e_UgridPowerMode := eUgridPowermode.None;
		END_CASE
	
		CASE WordEndian(Input.ui_Earthingsystem) OF
			//0: remain
			1:	get.HardSettings.system.e_EarthingSystem := eEarthingSystems.TN ; 
			2:	get.HardSettings.system.e_EarthingSystem := eEarthingSystems.IT ; 
		END_CASE
			
		CASE WordEndian(Input.GridConnectionMode) OF
			1:	get.SoftSettings.system.e_NetcontactorMode := eNetcontMode.auto; 
			2:	get.SoftSettings.system.e_NetcontactorMode := eNetcontMode.left;  
			3:	get.SoftSettings.system.e_NetcontactorMode := eNetcontMode.right; 
			4:	get.SoftSettings.system.e_NetcontactorMode := eNetcontMode.none; 
		ELSE
			get.SoftSettings.system.e_NetcontactorMode := eNetcontMode.auto; 	//Illegal input, return to auto
			//add diagnostic?
		END_CASE
		
		rtrig_disconnectNetcontactor(clk := (get.SoftSettings.system.e_NetcontactorMode = eNetcontMode.none) AND monitor.powerstack.Netcontactor.b_NetConFb);
		get.control.b_stop := rtrig_disconnectNetcontactor.q;
		
		ftrig_disconnectNetcontactor(clk := (get.SoftSettings.system.e_NetcontactorMode = eNetcontMode.none) AND NOT monitor.powerstack.Netcontactor.b_NetConFb);
		IF (monitor.powerstack.e_State = eStatusPowerstack.idle OR monitor.powerstack.e_State = eStatusPowerstack.GridCodeStop) THEN
			get.control.b_start := ftrig_disconnectNetcontactor.Q;
		END_IF
		
		
		Input.PrimaryDigOutState :=  WordEndian(Input.PrimaryDigOutState);
		IF Input.PrimaryDigOutState > 2 THEN
			Settings.MachineParams.HartingIO.PrimaryOutputContactSignal := Input.PrimaryDigOutState-3;
		ELSE
			IF Input.PrimaryDigOutState = 2 THEN	Settings.MachineParams.HartingIO.PrimaryOutputContactSignal := eOutputContactSignal.ManualClose; END_IF
			IF Input.PrimaryDigOutState = 1 THEN	Settings.MachineParams.HartingIO.PrimaryOutputContactSignal := eOutputContactSignal.ManualOpen; END_IF
		END_IF
			
		
		Input.SecondaryDigOutState :=  WordEndian(Input.SecondaryDigOutState);
		IF Input.SecondaryDigOutState > 2 THEN
			Settings.MachineParams.HartingIO.SecondaryOutputContactSignal := Input.SecondaryDigOutState-3;
		ELSE
			IF Input.SecondaryDigOutState = 2 THEN	Settings.MachineParams.HartingIO.SecondaryOutputContactSignal := eOutputContactSignal.ManualClose; END_IF
			IF Input.SecondaryDigOutState = 1 THEN	Settings.MachineParams.HartingIO.SecondaryOutputContactSignal := eOutputContactSignal.ManualOpen; END_IF
		END_IF
		
		IF  WordEndian(Input.PrimaryDigInState) > 0 THEN
			Settings.MachineParams.HartingIO.PrimaryInputContactSignal := WordEndian(Input.PrimaryDigInState)-1;
		END_IF
		
		IF  WordEndian(Input.SecondaryDigInState) > 0 THEN
			Settings.MachineParams.HartingIO.SecondaryInputContactSignal := WordEndian(Input.SecondaryDigInState)-1;
		END_IF
		
	END_IF
	

END_IF
END_METHOD

METHOD MapGeneratorControl : BOOL
VAR_IN_OUT CONSTANT
	monitor								: ST_System_Monitor;
END_VAR

VAR_IN_OUT
	events	: 	ST_ExtController_Events;
	Input	:	st_PNInput_GenControl;
	Output	:	ST_PNOutput_GenControl;
END_VAR
	
//Fill output data
Output.w_Status.0	:=	(monitor.system.GenGridController.b_extGensetMode OR
						monitor.system.GenGridController.e_BreakerMode = ebreakeroperationmode.GenIso OR
						monitor.system.GenGridController.e_BreakerMode = ebreakeroperationmode.GenFix OR
						monitor.system.GenGridController.e_BreakerMode = ebreakeroperationmode.GenDroop);
Output.w_Status.1	:= 	Output.w_Status.0 AND (monitor.system.GenGridController.e_state = eGenGridState.Cooldown OR 
						monitor.system.GenGridController.e_state = eGenGridState.Running OR
						monitor.system.GenGridController.e_state = eGenGridState.Warmup);
Output.w_Status		:= WordEndian(Output.w_Status);

Output.w_Warnings.0	:=	monitor.system.GenGridController.events.b_OverFreqTrip;
Output.w_Warnings.1	:=	monitor.system.GenGridController.events.b_UnderFreqTrip;
Output.w_Warnings.2	:=	monitor.system.GenGridController.events.b_OverloadTrip;
Output.w_Warnings.3	:=	monitor.system.GenGridController.events.b_ShutdownTimeOut;
Output.w_Warnings.4	:=	monitor.system.GenGridController.events.b_StartupFault;
Output.w_Warnings.5	:=	monitor.system.GenGridController.events.b_WarmupFault;
Output.w_Warnings.6	:=	monitor.system.GenGridController.events.b_GenDownTrip;
Output.w_Warnings		:= WordEndian(Output.w_Warnings);

Output.w_Faults		:= WordEndian(Output.w_Faults);

IF (monitor.system.GenGridController.b_extGensetMode OR
	monitor.system.GenGridController.e_BreakerMode = ebreakeroperationmode.GenIso OR
	monitor.system.GenGridController.e_BreakerMode = ebreakeroperationmode.GenFix OR
	monitor.system.GenGridController.e_BreakerMode = ebreakeroperationmode.GenDroop) THEN	
	
	CASE monitor.system.GenGridController.e_state OF
		eGenGridState.Waiting_Trigger:			Output.ui_GeneratorStatus := 1;
		eGenGridState.Starting:					Output.ui_GeneratorStatus := 2;
		eGenGridState.Warmup:					Output.ui_GeneratorStatus := 3;
		eGenGridState.Synchronization:			Output.ui_GeneratorStatus := 4;
		eGengridState.Running:					Output.ui_GeneratorStatus := 5;
		eGengridState.stopping:					Output.ui_GeneratorStatus := 6;
		eGengridState.Cooldown:					Output.ui_GeneratorStatus := 7;
	END_CASE
ELSE
	Output.ui_GeneratorStatus := 0;
END_IF
Output.ui_GeneratorStatus := WordEndian(Output.ui_GeneratorStatus);



//process input data, All inputs require Advancedcontrol
IF (NOT events.b_HeartbeatFault) AND ExternalControlMode = eExternalControlMode.AdvancedControl THEN
	input.w_Control := wordEndian(input.w_Control);
	get.SoftSettings.inputgenset.b_HydridMode 			:= input.w_Control.2;
	//3 was external genset. Now moved to general
	get.SoftSettings.inputgenset.b_FreqProtectionEnable	:=	input.w_Control.4;
	get.SoftSettings.setup.b_ExtGenset					:= Input.w_Control.3;
				
	UIntToReal(	in			:= Input.ui_SOCStart, 
				scale 		:= 10, 
				limitlow	:= 10,
				limithigh	:=	get.SoftSettings.inputgenset.setpointTimeslot1.r_SoCStop,
    			OutOfRange 	=>	,
				IgnoreZero 	:= TRUE,
				Out 		:= Get.SoftSettings.inputgenset.setpointTimeslot1.r_SoCStart );
	
	UIntToReal(	in			:= Input.ui_SOCStop, 
				scale 		:= 10, 
				limitlow	:= Get.SoftSettings.inputgenset.setpointTimeslot1.r_SoCStart,
				limithigh	:=	100,
    			OutOfRange 	=>	,
				IgnoreZero 	:= TRUE,
				Out 		:= Get.SoftSettings.inputgenset.setpointTimeslot1.r_SoCStop );
	
	UIntToReal(	in			:= Input.ui_BattLoadStart, 
				scale 		:= 10, 
				limitlow	:= 10,
				limithigh	:=	get.SoftSettings.inputgenset.setpointTimeslot1.r_BatteryloadStop,
    			OutOfRange 	=>	,
				IgnoreZero 	:= TRUE,
				Out 		:= Get.SoftSettings.inputgenset.setpointTimeslot1.r_BatteryloadStart );
	
	UIntToReal(	in			:= Input.ui_BattLoadStop, 
				scale 		:= 10, 
				limitlow	:= Get.SoftSettings.inputgenset.setpointTimeslot1.r_BatteryloadStart,
				limithigh	:=	100,
    			OutOfRange 	=>	,
				IgnoreZero 	:= TRUE,
				Out 		:= Get.SoftSettings.inputgenset.setpointTimeslot1.r_BatteryloadStop );
	
	CASE wordendian(input.ui_GenPowerMode) OF
		1:	get.SoftSettings.inputgenset.Generator.e_GensetMode := eGensetmode.Isochronous;
		2:	get.SoftSettings.inputgenset.Generator.e_GensetMode := eGensetmode.Droop;
		3:	get.SoftSettings.inputgenset.Generator.e_GensetMode := eGensetmode.FixedPower;		
	END_CASE
	
	UIntToReal(	in			:= Input.ui_GenRatedPower, 
				scale 		:= 1, 
				limitlow	:= 0,
				limithigh	:=	1000,
    			OutOfRange 	=>	,
				IgnoreZero 	:= TRUE,
				Out 		:= Get.SoftSettings.inputgenset.Generator.r_RatedPower );		
	
	UIntToReal(	in			:= Input.ui_GenMaxPowerLevel, 
				scale 		:= 10, 
				limitlow	:= get.SoftSettings.inputgenset.Generator.r_PowerloadMin,
				limithigh	:=	100,
    			OutOfRange 	=>	,
				IgnoreZero 	:= TRUE,
				Out 		:= Get.SoftSettings.inputgenset.Generator.r_powerloadMax );		
		
	UIntToReal(	in			:= Input.ui_GenEffPowerLevel, 
				scale 		:= 10, 
				limitlow	:= Get.SoftSettings.inputgenset.Generator.r_powerloadMin,
				limithigh	:= get.SoftSettings.inputgenset.Generator.r_powerloadMax,
    			OutOfRange 	=>	,
				IgnoreZero 	:= FALSE,
				Out 		:= Get.SoftSettings.inputgenset.Generator.r_powerloadEff );			
		
	UIntToReal(	in			:= Input.ui_GenMinPowerLevel, 
				scale 		:= 10, 
				limitlow	:= 0,
				limithigh	:= get.SoftSettings.inputgenset.Generator.r_powerloadMax,
    			OutOfRange 	=>	,
				IgnoreZero 	:= FALSE,
				Out 		:= Get.SoftSettings.inputgenset.Generator.r_powerloadMin );		
				
	get.SoftSettings.inputgenset.Generator.ui_WarmupTime					:=	wordEndian(Input.ui_GenWarmupTime);
	get.SoftSettings.inputgenset.Generator.ui_CooldownTime					:=	wordEndian(Input.ui_GenCooldownTime);
	get.SoftSettings.inputgenset.Generator.r_ramprate						:=	wordEndian(input.ui_IsoPowerRamp)/10;
	//get.Operation.Genset. //.ManualSetpoint									:=	wordEndian(Input.ui_GenCooldownTime);
	
	CASE WordEndian(Input.ui_StartStopControl) OF
		//0:	remain
		1:	get.SoftSettings.inputgenset.b_AutoStartStop := TRUE;
			get.Operation.Genset.b_manualStart := FALSE;
			
		2:	get.SoftSettings.inputgenset.b_AutoStartStop := FALSE;
			get.Operation.Genset.b_manualStart := FALSE;
			IF monitor.system.GenGridController.e_GensetStartStop = egensetstartstop.Stop THEN
 				get.Operation.Genset.b_manualStart := TRUE;
			END_IF
						
		3:	get.SoftSettings.inputgenset.b_AutoStartStop := FALSE;
			get.Operation.Genset.b_manualStart := FALSE;
			IF  monitor.system.GenGridController.e_GensetStartStop = egensetstartstop.Start THEN
				get.Operation.Genset.b_manualStart := TRUE;
			END_IF
	END_CASE
END_IF
END_METHOD

METHOD MapInputField : BOOL

VAR_IN_OUT CONSTANT
	monitor								: ST_System_Monitor;
END_VAR

VAR_IN_OUT
	events	: 	ST_ExtController_Events;
	Input	:	ST_PNInput_InputField;
	Output	:	ST_PNOutput_InputField;

END_VAR
//Fill output data
Output.w_Status.0	:=	Monitor.ACswitchgear.b_InputContactorfb;
Output.w_Status.1	:=	Monitor.ACswitchgear.b_InputMCCBfb;
Output.w_Status.2	:=	Monitor.ACswitchgear.b_InputSynchronizerfb;
Output.w_Status.8	:=	get.SoftSettings.setup.e_AcInputType = eACInputtype.None AND monitor.system.GenGridController.b_ModeChanged;
Output.w_Status.9	:=	get.SoftSettings.setup.e_AcInputType = eACInputtype.Genset AND monitor.system.GenGridController.b_ModeChanged;
Output.w_Status.10	:=	get.SoftSettings.setup.e_AcInputType = eACInputtype.Grid AND monitor.system.GenGridController.b_ModeChanged;
Output.w_Status.15	:= 	Monitor.ACswitchgear.b_InputSectionAvailable;
Output.w_Status		:= WordEndian(Output.w_Status);

//input overload warning toevoegen + heroverweeg indeling
Output.w_Warnings.0	:=	monitor.system.GenGridController.events.b_RotationFieldFault;
Output.w_Warnings.1	:=	monitor.system.GenGridController.events.b_CurrentLimitDisconnect;
Output.w_Warnings.2 :=	monitor.system.GenGridController.events.b_EmstopDisconnect;
Output.w_Warnings.3 :=	monitor.system.GenGridController.events.b_ShutdownDisconnect;
Output.w_Warnings.8 :=	monitor.system.GenGridController.events.b_TransToGenFixInhibit;
Output.w_Warnings.9 :=	monitor.system.GenGridController.events.b_TransToGenDroopInhibit;
Output.w_Warnings.10 :=	monitor.system.GenGridController.events.b_TransToGenIsoInhibit;
Output.w_Warnings	:= WordEndian(Output.w_Warnings);

Output.w_Faults.0	:=	monitor.system.GenGridController.events.b_OverloadTrip;
Output.w_Faults.1	:=	Monitor.powermonitor.events.b_MBCommError OR Monitor.powermonitor.events.b_EL3443Error;
Output.w_Faults.2	:= 	FALSE; //synchronizer fault. status doesn't exist yet?
Output.w_Faults.3	:= 	monitor.ACswitchgear.events.b_InputContactorFault;
Output.w_Faults		:= WordEndian(output.w_Faults);

	//not sure if this is the right variable
CASE wordendian(monitor.system.GenGridController.e_PowerControlMode) OF
	ePowerControlMode.None, ePowerControlMode.PeakshaveExt:
		output.ui_InputConnectionType := 1;
	ePowerControlMode.PeakshaveInputGrid:
		output.ui_InputConnectionType := 2;
	ePowerControlMode.PeakshaveInputGen:
		output.ui_InputConnectionType := 3;	
END_CASE
output.ui_InputConnectionType := wordendian(output.ui_InputConnectionType);

Output.i_ActivePower 			:=	RealToint (	In	:= Monitor.powermonitor.InputField.ar_ActivePower[0], 	Scale	:=	10);
Output.i_ReactivePower 			:=	RealToint (	In	:= Monitor.powermonitor.InputField.ar_ReactivePower[0], Scale	:=	10);
Output.i_PowerFactor 			:=	RealToint (	In	:= Monitor.powermonitor.InputField.ar_PowerFactor[0], Scale	:=	100);
Output.ui_frequency				:=	RealToUint(	In	:= Monitor.powermonitor.InputField.ar_Frequency[0], 	Scale	:=	10);
Output.ui_VoltageL1N			:=	RealToUint(	In	:= Monitor.powermonitor.InputField.ar_PhaseVoltage[1], Scale	:=	10);
Output.ui_VoltageL2N			:=	RealToUint(	In	:= Monitor.powermonitor.InputField.ar_PhaseVoltage[2], Scale	:=	10);
Output.ui_VoltageL3N			:=	RealToUint(	In	:= Monitor.powermonitor.InputField.ar_PhaseVoltage[3], Scale	:=	10);
Output.ui_VoltageL1L2			:=	RealToUint(	In	:= Monitor.powermonitor.InputField.ar_LineVoltage[1], Scale	:=	10);
Output.ui_VoltageL2L3			:=	RealToUint(	In	:= Monitor.powermonitor.InputField.ar_LineVoltage[2], Scale	:=	10);
Output.ui_VoltageL3L1			:=	RealToUint(	In	:= Monitor.powermonitor.InputField.ar_LineVoltage[3], Scale	:=	10);
Output.ui_CurrentL1				:=	RealToUint(	In	:= Monitor.powermonitor.InputField.ar_Current[1], 	Scale	:=	10);
Output.ui_CurrentL2				:=	RealToUint(	In	:= Monitor.powermonitor.InputField.ar_Current[2], 	Scale	:=	10);
Output.ui_CurrentL3				:=	RealToUint(	In	:= Monitor.powermonitor.InputField.ar_Current[3], 	Scale	:=	10);
Output.ui_CurrentN				:=	RealToUint(	In	:= Monitor.powermonitor.InputField.ar_Current[4], 	Scale	:=	10);
Output.ui_CurrentLimitField		:=	RealToUint( In	:= Monitor.Protections.OvercurrentProtection.r_TotalinputCurrentLimit, 	scale	:=	1);
Output.udi_TotalEnergyConsumed	:=	RealToUdint(In	:=	monitor.powermonitor.InputField.r_EnergyConsumed, Scale	:=	10);
Output.udi_TotalEnergySupplied	:= 	RealToUdint(In	:=	monitor.powermonitor.InputField.r_EnergySupplied, Scale	:=	10);

Output.ui_Current1L1			:=	RealToUint(	In	:= Monitor.powermonitor.InputField.Powerlock[1].ar_Current[1], 	Scale	:=	10);
Output.ui_Current1L2			:=	RealToUint(	In	:= Monitor.powermonitor.InputField.Powerlock[1].ar_Current[2], 	Scale	:=	10);
Output.ui_Current1L3			:=	RealToUint(	In	:= Monitor.powermonitor.InputField.Powerlock[1].ar_Current[3], 	Scale	:=	10);
Output.ui_Current1N				:=	RealToUint(	In	:= Monitor.powermonitor.InputField.Powerlock[1].ar_Current[4], 	Scale	:=	10);
Output.ui_Current2L1			:=	RealToUint(	In	:= Monitor.powermonitor.InputField.Powerlock[2].ar_Current[1], 	Scale	:=	10);
Output.ui_Current2L2			:=	RealToUint(	In	:= Monitor.powermonitor.InputField.Powerlock[2].ar_Current[2], 	Scale	:=	10);
Output.ui_Current2L3			:=	RealToUint(	In	:= Monitor.powermonitor.InputField.Powerlock[2].ar_Current[3], 	Scale	:=	10);
Output.ui_Current2N				:=	RealToUint(	In	:= Monitor.powermonitor.InputField.Powerlock[2].ar_Current[4], 	Scale	:=	10);

IF (NOT events.b_HeartbeatFault) AND ExternalControlMode > eExternalControlMode.BasicControl THEN
	Input.w_Control := WordEndian(input.w_Control);
	ManualAckState := Input.w_Control.0;
	
	CASE WordEndian(Input.InputConnectionType) OF
		//0:	remain
		1:	get.SoftSettings.setup.e_AcInputType := eAcInputType.None; 
		2:	get.SoftSettings.setup.e_AcInputType := eAcInputType.Grid;
		3:	get.SoftSettings.setup.e_AcInputType := eAcInputType.Genset; 
	END_CASE
	
	GenGridControllerStateMachine();
END_IF
END_METHOD

METHOD MapInputGridControl : BOOL
VAR_IN_OUT CONSTANT
	monitor								: ST_System_Monitor;
END_VAR

VAR_IN_OUT
	events	: 	ST_ExtController_Events;
	Input	:	st_PNInput_InputGridControl;
	Output	:	st_PNOutput_InputGridControl;
END_VAR

VAR_INST
	rtrig_openInputBreaker	:	r_trig;
	Rtrig_BreakerToAuto		:	r_trig;
	ftrig_ackDone			:	f_trig;
END_VAR
	
//Fill output data
Output.w_Status.0	:=	monitor.system.GenGridController.e_BreakerMode = eBreakerOperationMode.GridFeedthrough;
Output.w_Status		:= WordEndian(Output.w_Status);

Output.w_Warnings.0	:=	monitor.system.GenGridController.events.b_GridLostTrip; //?
Output.w_Warnings		:= WordEndian(Output.w_Warnings);

Output.w_Faults.0	:=	monitor.system.GenGridController.events.b_SynchronisationFault;
Output.w_Faults		:= 	WordEndian(Output.w_Faults);

//Output.ui_InputGridStatus := 0;
IF Output.w_Status.0 THEN	
	CASE monitor.system.GenGridController.e_state OF
		eGenGridState.Waiting_For_AC:			Output.ui_InputGridStatus := 1;
		eGenGridState.Waiting_Mode_Reconnect:	Output.ui_InputGridStatus := 2;
		eGenGridState.Gridcode_Release_Check:	Output.ui_InputGridStatus := 3;
		eGenGridState.Synchronization:			Output.ui_InputGridStatus := 4;
		eGengridState.Running:					Output.ui_InputGridStatus := 5;
		eGengridState.stopping:					Output.ui_InputGridStatus := 6;
	END_CASE
ELSE
	Output.ui_InputGridStatus := 0;
END_IF
Output.ui_InputGridStatus := wordendian(Output.ui_InputGridStatus);

IF (NOT events.b_HeartbeatFault) AND ExternalControlMode > eExternalControlMode.BasicControl AND monitor.system.GenGridController.e_BreakerMode = eBreakerOperationMode.GridFeedthrough THEN
	input.w_Control := wordEndian(input.w_Control);
	//get.SoftSettings.inputgrid.breaker.AutoConnect := input.w_Control.0;
	//get.Operation.inputgrid.b_SyncClose				:= input.w_Control.1;
	
	get.SoftSettings.system.b_AMF	 				:= input.w_Control.2;
	get.SoftSettings.inputgrid.b_GridCodesActive	:= NOT input.w_Control.3;
	
	IF input.w_Control.4 THEN
		get.SoftSettings.inputgrid.PeakshaveMode	:= 	ePeakShaveMode.Singlephase;
	ELSE
		get.SoftSettings.inputgrid.PeakshaveMode	:= 	ePeakShaveMode.Multiphase;		
	END_IF
	
	get.SoftSettings.inputgrid.Breaker.EMstopDisconnect		:= 	Input.w_Control.8;	//Maybe unneccessary to write both?
	get.SoftSettings.inputgrid.Breaker.ShutdownDisconnect	:= 	Input.w_Control.9;
	get.SoftSettings.inputgrid.Breaker.CurrentLimitDisconnect 	:=	Input.w_Control.10;
	
	UIntToReal(	in			:= Input.ui_FeedInCurrentLimit, 
				scale 		:= 10, 
				limitlow	:= 0,
				limithigh	:= 700,//get.HardSettings.inputgrid.r_FeedInCurrentLimitHard,
    			OutOfRange 	=>	,
				IgnoreZero 	:= FALSE,
				Out 		:= get.SoftSettings.inputgrid.setpointTimeslot1.r_FeedInCurrentLimitSoft );		

	UIntToReal(	in			:= Input.ui_SupplyCurrentLimit, 
				scale 		:= 10, 
				limitlow	:= 0,
				limithigh	:= 700,//get.HardSettings inputgrid.r_SupplyCurrentLimitHard,
    			OutOfRange 	=>	,
				IgnoreZero 	:= TRUE,
				Out 		:= get.SoftSettings.inputgrid.setpointTimeslot1.r_SupplyCurrentLimitSoft );		

	get.SoftSettings.inputgrid.breaker.CurrentLimitRetries := UINT_TO_BYTE(wordendian(input.ui_CurrentLimitRetries));	

	CASE wordEndian(input.ui_ContactorControl) OF
		1: get.SoftSettings.inputgrid.breaker.AutoConnect := TRUE;
		2: get.SoftSettings.inputgrid.breaker.AutoConnect := FALSE;
	END_CASE
END_IF
END_METHOD

METHOD MapOutputField : BOOL

VAR_IN_OUT CONSTANT
	monitor								: ST_System_Monitor;
END_VAR

VAR_IN_OUT
	Output	:	ST_PNOutput_OutputField;
END_VAR


//Fill output data
Output.w_Status.0	:=	Monitor.ACswitchgear.b_OutputMCCBfb;
Output.w_Status.1	:=	Monitor.ACswitchgear.b_PENlinkfb;
Output.w_Status.2	:= 	Monitor.powerstack.b_Gridtied;
Output.w_Status		:= WordEndian(Output.w_Status);

Output.w_Warnings.0	:=	Monitor.ACswitchgear.b_CEEprefuseOK;
Output.w_Warnings.1	:=	Monitor.ACswitchgear.b_OutputMCCBShuntOK;
Output.w_Warnings.2	:=	Monitor.powermonitor.events.b_MBCommWarning OR Monitor.powermonitor.events.b_MBTimeoutWarning;
Output.w_Warnings.3	:=	Monitor.protections.OvercurrentProtection.b_OutputWarning;
Output.w_Warnings	:= WordEndian(Output.w_Warnings);

Output.w_Faults.0	:=	Monitor.protections.OvercurrentProtection.b_OutputAlarm;
Output.w_Faults.1	:=	Monitor.powermonitor.events.b_MBCommError;
Output.w_Faults		:= WordEndian(output.w_Faults);

Output.i_ActivePower 			:=	RealToint (	In	:= Monitor.powermonitor.OutputField.ar_ActivePower[0], 	Scale	:=	10);
Output.i_ReactivePower 			:=	RealToint (	In	:= Monitor.powermonitor.OutputField.ar_ReactivePower[0], Scale	:=	10);
Output.i_PowerFactor 			:=	RealToint (	In	:= Monitor.powermonitor.OutputField.ar_PowerFactor[0], Scale	:=	100);
Output.ui_frequency				:=	RealToUint(	In	:= Monitor.powermonitor.OutputField.ar_Frequency[0] , 	Scale	:=	100);
Output.ui_VoltageL1N			:=	RealToUint(	In	:= Monitor.powermonitor.OutputField.ar_PhaseVoltage[1], Scale:=	10);
Output.ui_VoltageL2N			:=	RealToUint(	In	:= Monitor.powermonitor.OutputField.ar_PhaseVoltage[2], Scale:=	10);
Output.ui_VoltageL3N			:=	RealToUint(	In	:= Monitor.powermonitor.OutputField.ar_PhaseVoltage[3], Scale:=	10);
Output.ui_VoltageL1L2			:=	RealToUint(	In	:= Monitor.powermonitor.OutputField.ar_LineVoltage[1], Scale	:=	10);
Output.ui_VoltageL2L3			:=	RealToUint(	In	:= Monitor.powermonitor.OutputField.ar_LineVoltage[2], Scale	:=	10);
Output.ui_VoltageL3L1			:=	RealToUint(	In	:= Monitor.powermonitor.OutputField.ar_LineVoltage[3], Scale	:=	10);
Output.ui_CurrentL1				:=	RealToUint(	In	:= Monitor.powermonitor.OutputField.ar_Current[1], 	Scale	:=	10);
Output.ui_CurrentL2				:=	RealToUint(	In	:= Monitor.powermonitor.OutputField.ar_Current[2], 	Scale	:=	10);
Output.ui_CurrentL3				:=	RealToUint(	In	:= Monitor.powermonitor.OutputField.ar_Current[3], 	Scale	:=	10);
Output.ui_CurrentN				:=	RealToUint(	In	:= Monitor.powermonitor.OutputField.ar_Current[4], 	Scale	:=	10);
Output.ui_CurrentLimitField		:=	RealToUint (In	:= Monitor.Protections.OvercurrentProtection.r_TotalOutputCurrentLimit, 	scale	:=	1);
Output.udi_TotalEnergyConsumed	:= RealToUdint(	In	:=	monitor.powermonitor.OutputField.r_EnergyConsumed, Scale	:=	10);
Output.udi_TotalEnergySupplied	:= RealToUdint(	In	:=	monitor.powermonitor.OutputField.r_EnergySupplied, Scale	:=	10);

Output.ui_Current1L1			:=	RealToUint(	In	:= Monitor.powermonitor.OutputField.Powerlock[1].ar_Current[1], 	Scale	:=	10);
Output.ui_Current1L2			:=	RealToUint(	In	:= Monitor.powermonitor.OutputField.Powerlock[1].ar_Current[2], 	Scale	:=	10);
Output.ui_Current1L3			:=	RealToUint(	In	:= Monitor.powermonitor.OutputField.Powerlock[1].ar_Current[3], 	Scale	:=	10);
Output.ui_Current1N				:=	RealToUint(	In	:= Monitor.powermonitor.OutputField.Powerlock[1].ar_Current[4], 	Scale	:=	10);
Output.ui_Current2L1			:=	RealToUint(	In	:= Monitor.powermonitor.OutputField.Powerlock[2].ar_Current[1], 	Scale	:=	10);
Output.ui_Current2L2			:=	RealToUint(	In	:= Monitor.powermonitor.OutputField.Powerlock[2].ar_Current[2], 	Scale	:=	10);
Output.ui_Current2L3			:=	RealToUint(	In	:= Monitor.powermonitor.OutputField.Powerlock[2].ar_Current[3], 	Scale	:=	10);
Output.ui_Current2N				:=	RealToUint(	In	:= Monitor.powermonitor.OutputField.Powerlock[2].ar_Current[4], 	Scale	:=	10);
Output.ui_Current3L1			:=	RealToUint(	In	:= Monitor.powermonitor.OutputField.Powerlock[3].ar_Current[1], 	Scale	:=	10);
Output.ui_Current3L2			:=	RealToUint(	In	:= Monitor.powermonitor.OutputField.Powerlock[3].ar_Current[2], 	Scale	:=	10);
Output.ui_Current3L3			:=	RealToUint(	In	:= Monitor.powermonitor.OutputField.Powerlock[3].ar_Current[3], 	Scale	:=	10);
Output.ui_Current3N				:=	RealToUint(	In	:= Monitor.powermonitor.OutputField.Powerlock[3].ar_Current[4], 	Scale	:=	10);
END_METHOD

METHOD MapPeakShaveBox : BOOL
VAR_IN_OUT CONSTANT
	monitor								: ST_System_Monitor;
END_VAR

VAR_IN_OUT
	events	: 	ST_ExtController_Events;
	Input	:	ST_PNInput_Peakshavebox;
	Output	:	ST_PNOutput_Peakshavebox;
END_VAR
	
Output.w_Status.0	:=	Monitor.peakshavebox.b_buscouplerReady;
Output.w_Status.1	:= 	Monitor.peakshavebox.b_DataOK;
Output.w_Status.14	:=	Monitor.peakshavebox.b_active;
Output.w_Status.15	:= settings.Configuration.b_PeakshaverBoxEnable;//	Monitor.controlfb.softSettings.setup.b_peakshaveboxEnable;
Output.w_Status		:= WordEndian(Output.w_Status);

Output.w_Warnings.0	:= NOT Monitor.peakshavebox.b_dataOK;
output.w_Warnings.1 := Monitor.peakshavebox.b_SettingsChangePending;
Output.w_Warnings	:= WordEndian(Output.w_Warnings);

Output.w_Faults.0	:=	Monitor.peakshavebox.PowerStatus.b_Fault 
						OR Monitor.peakshavebox.PowerStatus.b_OverCurrent
						OR Monitor.peakshavebox.PowerStatus.b_OverVoltage
						OR Monitor.peakshavebox.PowerStatus.b_UnderVoltage;
Output.w_Faults		:= WordEndian(Output.w_Faults);

Output.i_ActivePower 		:=	RealToint (	In	:= 	Monitor.peakshavebox.Powermonitor.ar_ActivePower[0], 	scale := 10);												
Output.i_ReactivePower 		:=	RealToint (	In	:= 	Monitor.peakshavebox.Powermonitor.ar_ReactivePower[0], scale := 10);
Output.i_PowerFactor 		:=	RealToint (	In	:= Monitor.peakshavebox.Powermonitor.ar_PowerFactor[0], Scale	:=	100);													
Output.ui_frequency			:=	RealToUint(	In	:= Monitor.peakshavebox.Powermonitor.ar_Frequency[0], 		Scale	:=	10);
Output.ui_VoltageL1N		:=	RealToUint(	In	:= Monitor.peakshavebox.Powermonitor.ar_LineVoltage[1], 	Scale	:=	10);
Output.ui_VoltageL2N		:=	RealToUint(	In	:= Monitor.peakshavebox.Powermonitor.ar_LineVoltage[2], 	Scale	:=	10);
Output.ui_VoltageL3N		:=	RealToUint(	In	:= Monitor.peakshavebox.Powermonitor.ar_LineVoltage[3], 	Scale	:=	10);
Output.ui_VoltageL1L2		:=	RealToUint(	In	:= Monitor.peakshavebox.Powermonitor.ar_PhaseVoltage[1], 	Scale	:=	10);
Output.ui_VoltageL2L3		:=	RealToUint(	In	:= Monitor.peakshavebox.Powermonitor.ar_PhaseVoltage[2], 	Scale	:=	10);
Output.ui_VoltageL3L1		:=	RealToUint(	In	:= Monitor.peakshavebox.Powermonitor.ar_PhaseVoltage[3], 	Scale	:=	10);
Output.ui_CurrentL1			:=	RealToUint(	In	:= Monitor.peakshavebox.Powermonitor.ar_Current[1], 		Scale	:=	10);
Output.ui_CurrentL2			:=	RealToUint(	In	:= Monitor.peakshavebox.Powermonitor.ar_Current[2], 		Scale	:=	10);
Output.ui_CurrentL3			:=	RealToUint(	In	:= Monitor.peakshavebox.Powermonitor.ar_Current[3], 		Scale	:=	10);
Output.ui_CurrentN			:=	RealToUint(	In	:= Monitor.peakshavebox.Powermonitor.ar_Current[4], 		Scale	:=	10);


IF (NOT events.b_HeartbeatFault) AND ExternalControlMode > eExternalControlMode.BasicControl THEN
	input.w_Control := wordEndian(input.w_Control);
	get.SoftSettings.setup.b_PeakshaveBoxEnable := 	input.w_Control.0;
	get.SoftSettings.PSB.b_ReverseCTDirection	:=	input.w_Control.1;

	IF input.w_Control.2 THEN
		get.SoftSettings.PSB.PeakshaveMode	:= 	ePeakShaveMode.Singlephase;
	ELSE
		get.SoftSettings.PSB.PeakshaveMode	:= 	ePeakShaveMode.Multiphase;		
	END_IF
	
	UIntToReal(	in			:= Input.ui_FeedInCurrentLimit, 
				scale 		:= 10, 
				limitlow	:= 0,
				limithigh	:= st_params.limits.r_PSBCtLimit,
    			OutOfRange 	=>	events.b_PSBFeedInLimitOutOfRange,
				IgnoreZero 	:= FALSE,
				Out 		:= get.SoftSettings.PSB.setpointTimeslot1.r_FeedInCurrentLimitSoft );		

	UIntToReal(	in			:= Input.ui_SupplyCurrentLimit, 
				scale 		:= 10, 
				limitlow	:= 0,
				limithigh	:= st_params.limits.r_PSBCtLimit,
    			OutOfRange 	=>	events.b_PSBSupplyLimitOutOfRange,
				IgnoreZero 	:= TRUE,
				Out 		:= get.SoftSettings.PSB.setpointTimeslot1.r_SupplyCurrentLimitSoft );
	
	IF wordEndian(input.ui_VTRatio) > 0 THEN
		UIntToReal(	in			:= Input.ui_VTRatio, 
					scale 		:= 100, 
					limitlow	:= 0,
					limithigh	:= 655.35,
					OutOfRange 	=> ,
					IgnoreZero 	:= TRUE,
					Out 		:= get.SoftSettings.PSB.r_VTratio );	
	END_IF

	input.UI_CTRatio := wordEndian(input.UI_CTRatio);
	IF input.UI_CTRatio > 0 THEN		
		get.SoftSettings.PSB.ui_CTrange := input.UI_CTRatio;
	END_IF
END_IF
END_METHOD

METHOD MapPowerSTack : BOOL
VAR_IN_OUT CONSTANT
	monitor								: ST_System_Monitor;
END_VAR

